// TIA Portal V20 export
FUNCTION_BLOCK "Sequence_1_SemiAutoSplice"   // FB233, LAD
AUTHOR : ERsystem_FA2_DH. Kim
// stored: IsIECCheckEnabled true, MemoryReserve 100, Namespace Unit1.Em2, SetENOAutomatically false
   VAR
      statSelectedJobNumber { ExternalWritable := 'False'} : DInt;   // Evaluated Job Number
      instSequenceLADStatus { ExternalWritable := 'False'} : "LAF_StatusLadSequence";
      instSequenceLADControl { ExternalWritable := 'False'} : "LAF_ControlLadSequence";
      RetryCnt { S7_SetPoint := 'True'} : Array[0..9] of UInt;
      statPulse { ExternalWritable := 'False'} : Array[0..999] of Bool;
      statTonTimer { ExternalWritable := 'False'} : Array[0..9999] of TON_TIME;
   END_VAR
   VAR CONSTANT
      STEP_IDLE : DInt := 1;
      STEP_IMMEDIATE_STOP : DInt := 9001;   // Step executed when an immediate stop command is triggered for the sequence (i.e. when unit is in state aborting)
      SeqDelayTime : Time := T#100ms;
      SeqNoDelayTime : Time;
      RetrySV : UInt := 3;
      JOB_1_STEP_00 : DInt := 100;
      JOB_1_STEP_01 : DInt := 101;
      JOB_1_STEP_02 : DInt := 102;
      JOB_1_STEP_03 : DInt := 103;
      JOB_1_STEP_04 : DInt := 104;
      JOB_1_STEP_05 : DInt := 105;
      JOB_1_STEP_06 : DInt := 106;
      JOB_1_STEP_07 : DInt := 107;
      JOB_1_STEP_08 : DInt := 108;
      JOB_1_STEP_09 : DInt := 109;
      JOB_1_STEP_10 : DInt := 110;
      JOB_1_STEP_11 : DInt := 111;
      JOB_1_STEP_12 : DInt := 112;
      JOB_1_STEP_13 : DInt := 113;
      JOB_1_STEP_14 : DInt := 114;
      JOB_1_STEP_15 : DInt := 115;
      JOB_1_STEP_16 : DInt := 116;
      JOB_1_STEP_17 : DInt := 117;
      JOB_1_STEP_18 : DInt := 118;
      JOB_1_STEP_19 : DInt := 119;
      JOB_1_STEP_20 : DInt := 120;
      JOB_1_STEP_90 : DInt := 190;
      JOB_2_STEP_00 : DInt := 200;
      JOB_2_STEP_01 : DInt := 201;
      JOB_2_STEP_02 : DInt := 202;
      JOB_2_STEP_03 : DInt := 203;
      JOB_2_STEP_04 : DInt := 204;
      JOB_2_STEP_05 : DInt := 205;
      JOB_2_STEP_06 : DInt := 206;
      JOB_2_STEP_07 : DInt := 207;
      JOB_2_STEP_08 : DInt := 208;
      JOB_2_STEP_09 : DInt := 209;
      JOB_2_STEP_10 : DInt := 210;
      JOB_2_STEP_11 : DInt := 211;
      JOB_2_STEP_12 : DInt := 212;
      JOB_2_STEP_13 : DInt := 213;
      JOB_2_STEP_14 : DInt := 214;
      JOB_2_STEP_15 : DInt := 215;
      JOB_2_STEP_16 : DInt := 216;
      JOB_2_STEP_17 : DInt := 217;
      JOB_2_STEP_18 : DInt := 218;
      JOB_2_STEP_19 : DInt := 219;
      JOB_2_STEP_20 : DInt := 220;
      JOB_2_STEP_90 : DInt := 290;
      JOB_3_STEP_00 : DInt := 300;
      JOB_3_STEP_01 : DInt := 301;
      JOB_3_STEP_02 : DInt := 302;
      JOB_3_STEP_03 : DInt := 303;
      JOB_3_STEP_04 : DInt := 304;
      JOB_3_STEP_05 : DInt := 305;
      JOB_3_STEP_06 : DInt := 306;
      JOB_3_STEP_07 : DInt := 307;
      JOB_3_STEP_08 : DInt := 308;
      JOB_3_STEP_09 : DInt := 309;
      JOB_3_STEP_10 : DInt := 310;
      JOB_3_STEP_11 : DInt := 311;
      JOB_3_STEP_12 : DInt := 312;
      JOB_3_STEP_13 : DInt := 313;
      JOB_3_STEP_14 : DInt := 314;
      JOB_3_STEP_15 : DInt := 315;
      JOB_3_STEP_16 : DInt := 316;
      JOB_3_STEP_17 : DInt := 317;
      JOB_3_STEP_18 : DInt := 318;
      JOB_3_STEP_19 : DInt := 319;
      JOB_3_STEP_20 : DInt := 320;
      JOB_3_STEP_90 : DInt := 390;
      JOB_4_STEP_00 : DInt := 400;
      JOB_4_STEP_01 : DInt := 401;
      JOB_4_STEP_02 : DInt := 402;
      JOB_4_STEP_03 : DInt := 403;
      JOB_4_STEP_04 : DInt := 404;
      JOB_4_STEP_05 : DInt := 405;
      JOB_4_STEP_06 : DInt := 406;
      JOB_4_STEP_07 : DInt := 407;
      JOB_4_STEP_08 : DInt := 408;
      JOB_4_STEP_09 : DInt := 409;
      JOB_4_STEP_10 : DInt := 410;
      JOB_4_STEP_11 : DInt := 411;
      JOB_4_STEP_12 : DInt := 412;
      JOB_4_STEP_13 : DInt := 413;
      JOB_4_STEP_14 : DInt := 414;
      JOB_4_STEP_15 : DInt := 415;
      JOB_4_STEP_16 : DInt := 416;
      JOB_4_STEP_17 : DInt := 417;
      JOB_4_STEP_18 : DInt := 418;
      JOB_4_STEP_19 : DInt := 419;
      JOB_4_STEP_20 : DInt := 420;
      JOB_4_STEP_50 : DInt := 450;
      JOB_5_STEP_00 : DInt := 500;
      JOB_5_STEP_01 : DInt := 501;
      JOB_5_STEP_02 : DInt := 502;
      JOB_5_STEP_03 : DInt := 503;
      JOB_5_STEP_04 : DInt := 504;
      JOB_5_STEP_05 : DInt := 505;
      JOB_5_STEP_06 : DInt := 506;
      JOB_5_STEP_07 : DInt := 507;
      JOB_5_STEP_08 : DInt := 508;
      JOB_5_STEP_09 : DInt := 509;
      JOB_5_STEP_10 : DInt := 510;
      JOB_5_STEP_11 : DInt := 511;
      JOB_5_STEP_12 : DInt := 512;
      JOB_5_STEP_13 : DInt := 513;
      JOB_5_STEP_14 : DInt := 514;
      JOB_5_STEP_15 : DInt := 515;
      JOB_5_STEP_16 : DInt := 516;
      JOB_5_STEP_17 : DInt := 517;
      JOB_5_STEP_18 : DInt := 518;
      JOB_5_STEP_19 : DInt := 519;
      JOB_5_STEP_20 : DInt := 520;
      JOB_5_STEP_50 : DInt := 550;
      JOB_6_STEP_00 : DInt := 600;
      JOB_6_STEP_01 : DInt := 601;
      JOB_6_STEP_02 : DInt := 602;
      JOB_6_STEP_03 : DInt := 603;
      JOB_6_STEP_04 : DInt := 604;
      JOB_6_STEP_05 : DInt := 605;
      JOB_6_STEP_06 : DInt := 606;
      JOB_6_STEP_07 : DInt := 607;
      JOB_6_STEP_08 : DInt := 608;
      JOB_6_STEP_09 : DInt := 609;
      JOB_6_STEP_10 : DInt := 610;
      JOB_6_STEP_11 : DInt := 611;
      JOB_6_STEP_12 : DInt := 612;
      JOB_6_STEP_13 : DInt := 613;
      JOB_6_STEP_14 : DInt := 614;
      JOB_6_STEP_15 : DInt := 615;
      JOB_6_STEP_16 : DInt := 616;
      JOB_6_STEP_17 : DInt := 617;
      JOB_6_STEP_18 : DInt := 618;
      JOB_6_STEP_19 : DInt := 619;
      JOB_6_STEP_20 : DInt := 620;
      JOB_6_STEP_50 : DInt := 650;
      JOB_7_STEP_00 : DInt := 700;
      JOB_7_STEP_01 : DInt := 701;
      JOB_7_STEP_02 : DInt := 702;
      JOB_7_STEP_03 : DInt := 703;
      JOB_7_STEP_04 : DInt := 704;
      JOB_7_STEP_05 : DInt := 705;
      JOB_7_STEP_06 : DInt := 706;
      JOB_7_STEP_07 : DInt := 707;
      JOB_7_STEP_08 : DInt := 708;
      JOB_7_STEP_09 : DInt := 709;
      JOB_7_STEP_10 : DInt := 710;
      JOB_7_STEP_11 : DInt := 711;
      JOB_7_STEP_12 : DInt := 712;
      JOB_7_STEP_13 : DInt := 713;
      JOB_7_STEP_14 : DInt := 714;
      JOB_7_STEP_15 : DInt := 715;
      JOB_7_STEP_16 : DInt := 716;
      JOB_7_STEP_17 : DInt := 717;
      JOB_7_STEP_18 : DInt := 718;
      JOB_7_STEP_19 : DInt := 719;
      JOB_7_STEP_20 : DInt := 720;
      JOB_7_STEP_50 : DInt := 750;
      JOB_8_STEP_00 : DInt := 800;
      JOB_8_STEP_01 : DInt := 801;
      JOB_8_STEP_02 : DInt := 802;
      JOB_8_STEP_03 : DInt := 803;
      JOB_8_STEP_04 : DInt := 804;
      JOB_8_STEP_05 : DInt := 805;
      JOB_8_STEP_06 : DInt := 806;
      JOB_8_STEP_07 : DInt := 807;
      JOB_8_STEP_08 : DInt := 808;
      JOB_8_STEP_09 : DInt := 809;
      JOB_8_STEP_10 : DInt := 810;
      JOB_8_STEP_11 : DInt := 811;
      JOB_8_STEP_12 : DInt := 812;
      JOB_8_STEP_13 : DInt := 813;
      JOB_8_STEP_14 : DInt := 814;
      JOB_8_STEP_15 : DInt := 815;
      JOB_8_STEP_16 : DInt := 816;
      JOB_8_STEP_17 : DInt := 817;
      JOB_8_STEP_18 : DInt := 818;
      JOB_8_STEP_19 : DInt := 819;
      JOB_8_STEP_20 : DInt := 820;
      JOB_8_STEP_50 : DInt := 850;
      JOB_9_STEP_00 : DInt := 900;
      JOB_9_STEP_01 : DInt := 901;
      JOB_9_STEP_02 : DInt := 902;
      JOB_9_STEP_03 : DInt := 903;
      JOB_9_STEP_04 : DInt := 904;
      JOB_9_STEP_05 : DInt := 905;
      JOB_9_STEP_06 : DInt := 906;
      JOB_9_STEP_07 : DInt := 907;
      JOB_9_STEP_08 : DInt := 908;
      JOB_9_STEP_09 : DInt := 909;
      JOB_9_STEP_10 : DInt := 910;
      JOB_9_STEP_11 : DInt := 911;
      JOB_9_STEP_12 : DInt := 912;
      JOB_9_STEP_13 : DInt := 913;
      JOB_9_STEP_14 : DInt := 914;
      JOB_9_STEP_15 : DInt := 915;
      JOB_9_STEP_16 : DInt := 916;
      JOB_9_STEP_17 : DInt := 917;
      JOB_9_STEP_18 : DInt := 918;
      JOB_9_STEP_19 : DInt := 919;
      JOB_9_STEP_20 : DInt := 920;
      JOB_8_STEP_51 : DInt := 950;
      JOB_10_STEP_00 : DInt := 1000;
      JOB_10_STEP_01 : DInt := 1001;
      JOB_10_STEP_02 : DInt := 1002;
      JOB_10_STEP_03 : DInt := 1003;
      JOB_10_STEP_04 : DInt := 1004;
      JOB_10_STEP_05 : DInt := 1005;
      JOB_10_STEP_06 : DInt := 1006;
      JOB_10_STEP_07 : DInt := 1007;
      JOB_10_STEP_08 : DInt := 1008;
      JOB_10_STEP_09 : DInt := 1009;
      JOB_10_STEP_10 : DInt := 1010;
      JOB_10_STEP_11 : DInt := 1011;
      JOB_10_STEP_12 : DInt := 1012;
      JOB_10_STEP_13 : DInt := 1013;
      JOB_10_STEP_14 : DInt := 1014;
      JOB_10_STEP_15 : DInt := 1015;
      JOB_10_STEP_16 : DInt := 1016;
      JOB_10_STEP_17 : DInt := 1017;
      JOB_10_STEP_18 : DInt := 1018;
      JOB_10_STEP_19 : DInt := 1019;
      JOB_10_STEP_20 : DInt := 1020;
      JOB_10_STEP_50 : DInt := 1050;
      JOB_11_STEP_00 : DInt := 1100;
      JOB_11_STEP_01 : DInt := 1101;
      JOB_11_STEP_02 : DInt := 1102;
      JOB_11_STEP_03 : DInt := 1103;
      JOB_11_STEP_04 : DInt := 1104;
      JOB_11_STEP_05 : DInt := 1105;
      JOB_11_STEP_06 : DInt := 1106;
      JOB_11_STEP_07 : DInt := 1107;
      JOB_11_STEP_08 : DInt := 1108;
      JOB_11_STEP_09 : DInt := 1109;
      JOB_11_STEP_10 : DInt := 1110;
      JOB_11_STEP_11 : DInt := 1111;
      JOB_11_STEP_12 : DInt := 1112;
      JOB_11_STEP_13 : DInt := 1113;
      JOB_11_STEP_14 : DInt := 1114;
      JOB_11_STEP_15 : DInt := 1115;
      JOB_11_STEP_16 : DInt := 1116;
      JOB_11_STEP_17 : DInt := 1117;
      JOB_11_STEP_18 : DInt := 1118;
      JOB_11_STEP_19 : DInt := 1119;
      JOB_11_STEP_20 : DInt := 1120;
      JOB_11_STEP_50 : DInt := 1150;
      JOB_12_STEP_00 : DInt := 1200;
      JOB_12_STEP_01 : DInt := 1201;
      JOB_12_STEP_02 : DInt := 1202;
      JOB_12_STEP_03 : DInt := 1203;
      JOB_12_STEP_04 : DInt := 1204;
      JOB_12_STEP_05 : DInt := 1205;
      JOB_12_STEP_06 : DInt := 1206;
      JOB_12_STEP_07 : DInt := 1207;
      JOB_12_STEP_08 : DInt := 1208;
      JOB_12_STEP_09 : DInt := 1209;
      JOB_12_STEP_10 : DInt := 1210;
      JOB_12_STEP_11 : DInt := 1211;
      JOB_12_STEP_12 : DInt := 1212;
      JOB_12_STEP_13 : DInt := 1213;
      JOB_12_STEP_14 : DInt := 1214;
      JOB_12_STEP_15 : DInt := 1215;
      JOB_12_STEP_16 : DInt := 1216;
      JOB_12_STEP_17 : DInt := 1217;
      JOB_12_STEP_18 : DInt := 1218;
      JOB_12_STEP_19 : DInt := 1219;
      JOB_12_STEP_20 : DInt := 1220;
      JOB_12_STEP_50 : DInt := 1250;
      JOB_13_STEP_00 : DInt := 1300;
      JOB_13_STEP_01 : DInt := 1301;
      JOB_13_STEP_02 : DInt := 1302;
      JOB_13_STEP_03 : DInt := 1303;
      JOB_13_STEP_04 : DInt := 1304;
      JOB_13_STEP_05 : DInt := 1305;
      JOB_13_STEP_06 : DInt := 1306;
      JOB_13_STEP_07 : DInt := 1307;
      JOB_13_STEP_08 : DInt := 1308;
      JOB_13_STEP_09 : DInt := 1309;
      JOB_13_STEP_10 : DInt := 1310;
      JOB_13_STEP_11 : DInt := 1311;
      JOB_13_STEP_12 : DInt := 1312;
      JOB_13_STEP_13 : DInt := 1313;
      JOB_13_STEP_14 : DInt := 1314;
      JOB_13_STEP_15 : DInt := 1315;
      JOB_13_STEP_16 : DInt := 1316;
      JOB_13_STEP_17 : DInt := 1317;
      JOB_13_STEP_18 : DInt := 1318;
      JOB_13_STEP_19 : DInt := 1319;
      JOB_13_STEP_20 : DInt := 1320;
      JOB_13_STEP_50 : DInt := 1350;
      JOB_14_STEP_00 : DInt := 1400;
      JOB_14_STEP_01 : DInt := 1401;
      JOB_14_STEP_02 : DInt := 1402;
      JOB_14_STEP_03 : DInt := 1403;
      JOB_14_STEP_04 : DInt := 1404;
      JOB_14_STEP_05 : DInt := 1405;
      JOB_14_STEP_06 : DInt := 1406;
      JOB_14_STEP_07 : DInt := 1407;
      JOB_14_STEP_08 : DInt := 1408;
      JOB_14_STEP_09 : DInt := 1409;
      JOB_14_STEP_10 : DInt := 1410;
      JOB_14_STEP_11 : DInt := 1411;
      JOB_14_STEP_12 : DInt := 1412;
      JOB_14_STEP_13 : DInt := 1413;
      JOB_14_STEP_14 : DInt := 1414;
      JOB_14_STEP_15 : DInt := 1415;
      JOB_14_STEP_16 : DInt := 1416;
      JOB_14_STEP_17 : DInt := 1417;
      JOB_14_STEP_18 : DInt := 1418;
      JOB_14_STEP_19 : DInt := 1419;
      JOB_14_STEP_20 : DInt := 1420;
      JOB_14_STEP_50 : DInt := 1450;
      JOB_15_STEP_00 : DInt := 1500;
      JOB_15_STEP_01 : DInt := 1501;
      JOB_15_STEP_02 : DInt := 1502;
      JOB_15_STEP_03 : DInt := 1503;
      JOB_15_STEP_04 : DInt := 1504;
      JOB_15_STEP_05 : DInt := 1505;
      JOB_15_STEP_06 : DInt := 1506;
      JOB_15_STEP_07 : DInt := 1507;
      JOB_15_STEP_08 : DInt := 1508;
      JOB_15_STEP_09 : DInt := 1509;
      JOB_15_STEP_10 : DInt := 1510;
      JOB_15_STEP_11 : DInt := 1511;
      JOB_15_STEP_12 : DInt := 1512;
      JOB_15_STEP_13 : DInt := 1513;
      JOB_15_STEP_14 : DInt := 1514;
      JOB_15_STEP_15 : DInt := 1515;
      JOB_15_STEP_16 : DInt := 1516;
      JOB_15_STEP_17 : DInt := 1517;
      JOB_15_STEP_18 : DInt := 1518;
      JOB_15_STEP_19 : DInt := 1519;
      JOB_15_STEP_20 : DInt := 1520;
      JOB_15_STEP_50 : DInt := 1550;
      JOB_16_STEP_00 : DInt := 1600;
      JOB_16_STEP_01 : DInt := 1601;
      JOB_16_STEP_02 : DInt := 1602;
      JOB_16_STEP_03 : DInt := 1603;
      JOB_16_STEP_04 : DInt := 1604;
      JOB_16_STEP_05 : DInt := 1605;
      JOB_16_STEP_06 : DInt := 1606;
      JOB_16_STEP_07 : DInt := 1607;
      JOB_16_STEP_08 : DInt := 1608;
      JOB_16_STEP_09 : DInt := 1609;
      JOB_16_STEP_10 : DInt := 1610;
      JOB_16_STEP_11 : DInt := 1611;
      JOB_16_STEP_12 : DInt := 1612;
      JOB_16_STEP_13 : DInt := 1613;
      JOB_16_STEP_14 : DInt := 1614;
      JOB_16_STEP_15 : DInt := 1615;
      JOB_16_STEP_16 : DInt := 1616;
      JOB_16_STEP_17 : DInt := 1617;
      JOB_16_STEP_18 : DInt := 1618;
      JOB_16_STEP_19 : DInt := 1619;
      JOB_16_STEP_20 : DInt := 1620;
      JOB_16_STEP_50 : DInt := 1650;
      JOB_17_STEP_00 : DInt := 1700;
      JOB_17_STEP_01 : DInt := 1701;
      JOB_17_STEP_02 : DInt := 1702;
      JOB_17_STEP_03 : DInt := 1703;
      JOB_17_STEP_04 : DInt := 1704;
      JOB_17_STEP_05 : DInt := 1705;
      JOB_17_STEP_06 : DInt := 1706;
      JOB_17_STEP_07 : DInt := 1707;
      JOB_17_STEP_08 : DInt := 1708;
      JOB_17_STEP_09 : DInt := 1709;
      JOB_17_STEP_10 : DInt := 1710;
      JOB_17_STEP_11 : DInt := 1711;
      JOB_17_STEP_12 : DInt := 1712;
      JOB_17_STEP_13 : DInt := 1713;
      JOB_17_STEP_14 : DInt := 1714;
      JOB_17_STEP_15 : DInt := 1715;
      JOB_17_STEP_16 : DInt := 1716;
      JOB_17_STEP_17 : DInt := 1717;
      JOB_17_STEP_18 : DInt := 1718;
      JOB_17_STEP_19 : DInt := 1719;
      JOB_17_STEP_20 : DInt := 1720;
      JOB_17_STEP_50 : DInt := 1750;
      JOB_18_STEP_00 : DInt := 1800;
      JOB_18_STEP_01 : DInt := 1801;
      JOB_18_STEP_02 : DInt := 1802;
      JOB_18_STEP_03 : DInt := 1803;
      JOB_18_STEP_04 : DInt := 1804;
      JOB_18_STEP_05 : DInt := 1805;
      JOB_18_STEP_06 : DInt := 1806;
      JOB_18_STEP_07 : DInt := 1807;
      JOB_18_STEP_08 : DInt := 1808;
      JOB_18_STEP_09 : DInt := 1809;
      JOB_18_STEP_10 : DInt := 1810;
      JOB_18_STEP_11 : DInt := 1811;
      JOB_18_STEP_12 : DInt := 1812;
      JOB_18_STEP_13 : DInt := 1813;
      JOB_18_STEP_14 : DInt := 1814;
      JOB_18_STEP_15 : DInt := 1815;
      JOB_18_STEP_16 : DInt := 1816;
      JOB_18_STEP_17 : DInt := 1817;
      JOB_18_STEP_18 : DInt := 1818;
      JOB_18_STEP_19 : DInt := 1819;
      JOB_18_STEP_20 : DInt := 1820;
      JOB_18_STEP_50 : DInt := 1850;
      JOB_19_STEP_00 : DInt := 1900;
      JOB_19_STEP_01 : DInt := 1901;
      JOB_19_STEP_02 : DInt := 1902;
      JOB_19_STEP_03 : DInt := 1903;
      JOB_19_STEP_04 : DInt := 1904;
      JOB_19_STEP_05 : DInt := 1905;
      JOB_19_STEP_06 : DInt := 1906;
      JOB_19_STEP_07 : DInt := 1907;
      JOB_19_STEP_08 : DInt := 1908;
      JOB_19_STEP_09 : DInt := 1909;
      JOB_19_STEP_10 : DInt := 1910;
      JOB_19_STEP_11 : DInt := 1911;
      JOB_19_STEP_12 : DInt := 1912;
      JOB_19_STEP_13 : DInt := 1913;
      JOB_19_STEP_14 : DInt := 1914;
      JOB_19_STEP_15 : DInt := 1915;
      JOB_19_STEP_16 : DInt := 1916;
      JOB_19_STEP_17 : DInt := 1917;
      JOB_19_STEP_18 : DInt := 1918;
      JOB_19_STEP_19 : DInt := 1919;
      JOB_19_STEP_20 : DInt := 1920;
      JOB_19_STEP_50 : DInt := 1950;
      JOB_20_STEP_00 : DInt := 2000;
      JOB_20_STEP_01 : DInt := 2001;
      JOB_20_STEP_02 : DInt := 2002;
      JOB_20_STEP_03 : DInt := 2003;
      JOB_20_STEP_04 : DInt := 2004;
      JOB_20_STEP_05 : DInt := 2005;
      JOB_20_STEP_06 : DInt := 2006;
      JOB_20_STEP_07 : DInt := 2007;
      JOB_20_STEP_08 : DInt := 2008;
      JOB_20_STEP_09 : DInt := 2009;
      JOB_20_STEP_10 : DInt := 2010;
      JOB_20_STEP_11 : DInt := 2011;
      JOB_20_STEP_12 : DInt := 2012;
      JOB_20_STEP_13 : DInt := 2013;
      JOB_20_STEP_14 : DInt := 2014;
      JOB_20_STEP_15 : DInt := 2015;
      JOB_20_STEP_16 : DInt := 2016;
      JOB_20_STEP_17 : DInt := 2017;
      JOB_20_STEP_18 : DInt := 2018;
      JOB_20_STEP_19 : DInt := 2019;
      JOB_20_STEP_20 : DInt := 2020;
      JOB_20_STEP_50 : DInt := 2050;
      JOB_21_STEP_00 : DInt := 2100;
      JOB_21_STEP_01 : DInt := 2101;
      JOB_21_STEP_02 : DInt := 2102;
      JOB_21_STEP_03 : DInt := 2103;
      JOB_21_STEP_04 : DInt := 2104;
      JOB_21_STEP_05 : DInt := 2105;
      JOB_21_STEP_06 : DInt := 2106;
      JOB_21_STEP_07 : DInt := 2107;
      JOB_21_STEP_08 : DInt := 2108;
      JOB_21_STEP_09 : DInt := 2109;
      JOB_21_STEP_10 : DInt := 2110;
      JOB_21_STEP_11 : DInt := 2111;
      JOB_21_STEP_12 : DInt := 2112;
      JOB_21_STEP_13 : DInt := 2113;
      JOB_21_STEP_14 : DInt := 2114;
      JOB_21_STEP_15 : DInt := 2115;
      JOB_21_STEP_16 : DInt := 2116;
      JOB_21_STEP_17 : DInt := 2117;
      JOB_21_STEP_18 : DInt := 2118;
      JOB_21_STEP_19 : DInt := 2119;
      JOB_21_STEP_20 : DInt := 2120;
      JOB_21_STEP_50 : DInt := 2150;
      JOB_22_STEP_00 : DInt := 2200;
      JOB_22_STEP_01 : DInt := 2201;
      JOB_22_STEP_02 : DInt := 2202;
      JOB_22_STEP_03 : DInt := 2203;
      JOB_22_STEP_04 : DInt := 2204;
      JOB_22_STEP_05 : DInt := 2205;
      JOB_22_STEP_06 : DInt := 2206;
      JOB_22_STEP_07 : DInt := 2207;
      JOB_22_STEP_08 : DInt := 2208;
      JOB_22_STEP_09 : DInt := 2209;
      JOB_22_STEP_10 : DInt := 2210;
      JOB_22_STEP_11 : DInt := 2211;
      JOB_22_STEP_12 : DInt := 2212;
      JOB_22_STEP_13 : DInt := 2213;
      JOB_22_STEP_14 : DInt := 2214;
      JOB_22_STEP_15 : DInt := 2215;
      JOB_22_STEP_16 : DInt := 2216;
      JOB_22_STEP_17 : DInt := 2217;
      JOB_22_STEP_18 : DInt := 2218;
      JOB_22_STEP_19 : DInt := 2219;
      JOB_22_STEP_20 : DInt := 2220;
      JOB_22_STEP_50 : DInt := 2250;
      JOB_23_STEP_00 : DInt := 2300;
      JOB_23_STEP_01 : DInt := 2301;
      JOB_23_STEP_02 : DInt := 2302;
      JOB_23_STEP_03 : DInt := 2303;
      JOB_23_STEP_04 : DInt := 2304;
      JOB_23_STEP_05 : DInt := 2305;
      JOB_23_STEP_06 : DInt := 2306;
      JOB_23_STEP_07 : DInt := 2307;
      JOB_23_STEP_08 : DInt := 2308;
      JOB_23_STEP_09 : DInt := 2309;
      JOB_23_STEP_10 : DInt := 2310;
      JOB_23_STEP_11 : DInt := 2311;
      JOB_23_STEP_12 : DInt := 2312;
      JOB_23_STEP_13 : DInt := 2313;
      JOB_23_STEP_14 : DInt := 2314;
      JOB_23_STEP_15 : DInt := 2315;
      JOB_23_STEP_16 : DInt := 2316;
      JOB_23_STEP_17 : DInt := 2317;
      JOB_23_STEP_18 : DInt := 2318;
      JOB_23_STEP_19 : DInt := 2319;
      JOB_23_STEP_20 : DInt := 2320;
      JOB_23_STEP_50 : DInt := 2350;
      JOB_24_STEP_00 : DInt := 2400;
      JOB_24_STEP_01 : DInt := 2401;
      JOB_24_STEP_02 : DInt := 2402;
      JOB_24_STEP_03 : DInt := 2403;
      JOB_24_STEP_04 : DInt := 2404;
      JOB_24_STEP_05 : DInt := 2405;
      JOB_24_STEP_06 : DInt := 2406;
      JOB_24_STEP_07 : DInt := 2407;
      JOB_24_STEP_08 : DInt := 2408;
      JOB_24_STEP_09 : DInt := 2409;
      JOB_24_STEP_10 : DInt := 2410;
      JOB_24_STEP_11 : DInt := 2411;
      JOB_24_STEP_12 : DInt := 2412;
      JOB_24_STEP_13 : DInt := 2413;
      JOB_24_STEP_14 : DInt := 2414;
      JOB_24_STEP_15 : DInt := 2415;
      JOB_24_STEP_16 : DInt := 2416;
      JOB_24_STEP_17 : DInt := 2417;
      JOB_24_STEP_18 : DInt := 2418;
      JOB_24_STEP_19 : DInt := 2419;
      JOB_24_STEP_20 : DInt := 2420;
      JOB_24_STEP_50 : DInt := 2450;
      JOB_25_STEP_00 : DInt := 2500;
      JOB_25_STEP_01 : DInt := 2501;
      JOB_25_STEP_02 : DInt := 2502;
      JOB_25_STEP_03 : DInt := 2503;
      JOB_25_STEP_04 : DInt := 2504;
      JOB_25_STEP_05 : DInt := 2505;
      JOB_25_STEP_06 : DInt := 2506;
      JOB_25_STEP_07 : DInt := 2507;
      JOB_25_STEP_08 : DInt := 2508;
      JOB_25_STEP_09 : DInt := 2509;
      JOB_25_STEP_10 : DInt := 2510;
      JOB_25_STEP_11 : DInt := 2511;
      JOB_25_STEP_12 : DInt := 2512;
      JOB_25_STEP_13 : DInt := 2513;
      JOB_25_STEP_14 : DInt := 2514;
      JOB_25_STEP_15 : DInt := 2515;
      JOB_25_STEP_16 : DInt := 2516;
      JOB_25_STEP_17 : DInt := 2517;
      JOB_25_STEP_18 : DInt := 2518;
      JOB_25_STEP_19 : DInt := 2519;
      JOB_25_STEP_20 : DInt := 2520;
      JOB_25_STEP_50 : DInt := 2550;
      JOB_26_STEP_00 : DInt := 2600;
      JOB_26_STEP_01 : DInt := 2601;
      JOB_26_STEP_02 : DInt := 2602;
      JOB_26_STEP_03 : DInt := 2603;
      JOB_26_STEP_04 : DInt := 2604;
      JOB_26_STEP_05 : DInt := 2605;
      JOB_26_STEP_06 : DInt := 2606;
      JOB_26_STEP_07 : DInt := 2607;
      JOB_26_STEP_08 : DInt := 2608;
      JOB_26_STEP_09 : DInt := 2609;
      JOB_26_STEP_10 : DInt := 2610;
      JOB_26_STEP_11 : DInt := 2611;
      JOB_26_STEP_12 : DInt := 2612;
      JOB_26_STEP_13 : DInt := 2613;
      JOB_26_STEP_14 : DInt := 2614;
      JOB_26_STEP_15 : DInt := 2615;
      JOB_26_STEP_16 : DInt := 2616;
      JOB_26_STEP_17 : DInt := 2617;
      JOB_26_STEP_18 : DInt := 2618;
      JOB_26_STEP_19 : DInt := 2619;
      JOB_26_STEP_20 : DInt := 2620;
      JOB_26_STEP_50 : DInt := 2650;
      JOB_27_STEP_00 : DInt := 2700;
      JOB_27_STEP_01 : DInt := 2701;
      JOB_27_STEP_02 : DInt := 2702;
      JOB_27_STEP_03 : DInt := 2703;
      JOB_27_STEP_04 : DInt := 2704;
      JOB_27_STEP_05 : DInt := 2705;
      JOB_27_STEP_06 : DInt := 2706;
      JOB_27_STEP_07 : DInt := 2707;
      JOB_27_STEP_08 : DInt := 2708;
      JOB_27_STEP_09 : DInt := 2709;
      JOB_27_STEP_10 : DInt := 2710;
      JOB_27_STEP_11 : DInt := 2711;
      JOB_27_STEP_12 : DInt := 2712;
      JOB_27_STEP_13 : DInt := 2713;
      JOB_27_STEP_14 : DInt := 2714;
      JOB_27_STEP_15 : DInt := 2715;
      JOB_27_STEP_16 : DInt := 2716;
      JOB_27_STEP_17 : DInt := 2717;
      JOB_27_STEP_18 : DInt := 2718;
      JOB_27_STEP_19 : DInt := 2719;
      JOB_27_STEP_20 : DInt := 2720;
      JOB_27_STEP_50 : DInt := 2750;
      JOB_28_STEP_00 : DInt := 2800;
      JOB_28_STEP_01 : DInt := 2801;
      JOB_28_STEP_02 : DInt := 2802;
      JOB_28_STEP_03 : DInt := 2803;
      JOB_28_STEP_04 : DInt := 2804;
      JOB_28_STEP_05 : DInt := 2805;
      JOB_28_STEP_06 : DInt := 2806;
      JOB_28_STEP_07 : DInt := 2807;
      JOB_28_STEP_08 : DInt := 2808;
      JOB_28_STEP_09 : DInt := 2809;
      JOB_28_STEP_10 : DInt := 2810;
      JOB_28_STEP_11 : DInt := 2811;
      JOB_28_STEP_12 : DInt := 2812;
      JOB_28_STEP_13 : DInt := 2813;
      JOB_28_STEP_14 : DInt := 2814;
      JOB_28_STEP_15 : DInt := 2815;
      JOB_28_STEP_16 : DInt := 2816;
      JOB_28_STEP_17 : DInt := 2817;
      JOB_28_STEP_18 : DInt := 2818;
      JOB_28_STEP_19 : DInt := 2819;
      JOB_28_STEP_20 : DInt := 2820;
      JOB_28_STEP_50 : DInt := 2850;
      JOB_29_STEP_00 : DInt := 2900;
      JOB_29_STEP_01 : DInt := 2901;
      JOB_29_STEP_02 : DInt := 2902;
      JOB_29_STEP_03 : DInt := 2903;
      JOB_29_STEP_04 : DInt := 2904;
      JOB_29_STEP_05 : DInt := 2905;
      JOB_29_STEP_06 : DInt := 2906;
      JOB_29_STEP_07 : DInt := 2907;
      JOB_29_STEP_08 : DInt := 2908;
      JOB_29_STEP_09 : DInt := 2909;
      JOB_29_STEP_10 : DInt := 2910;
      JOB_29_STEP_11 : DInt := 2911;
      JOB_29_STEP_12 : DInt := 2912;
      JOB_29_STEP_13 : DInt := 2913;
      JOB_29_STEP_14 : DInt := 2914;
      JOB_29_STEP_15 : DInt := 2915;
      JOB_29_STEP_16 : DInt := 2916;
      JOB_29_STEP_17 : DInt := 2917;
      JOB_29_STEP_18 : DInt := 2918;
      JOB_29_STEP_19 : DInt := 2919;
      JOB_29_STEP_20 : DInt := 2920;
      JOB_29_STEP_50 : DInt := 2950;
      JOB_30_STEP_00 : DInt := 3000;
      JOB_30_STEP_01 : DInt := 3001;
      JOB_30_STEP_02 : DInt := 3002;
      JOB_30_STEP_03 : DInt := 3003;
      JOB_30_STEP_04 : DInt := 3004;
      JOB_30_STEP_05 : DInt := 3005;
      JOB_30_STEP_06 : DInt := 3006;
      JOB_30_STEP_07 : DInt := 3007;
      JOB_30_STEP_08 : DInt := 3008;
      JOB_30_STEP_09 : DInt := 3009;
      JOB_30_STEP_10 : DInt := 3010;
      JOB_30_STEP_11 : DInt := 3011;
      JOB_30_STEP_12 : DInt := 3012;
      JOB_30_STEP_13 : DInt := 3013;
      JOB_30_STEP_14 : DInt := 3014;
      JOB_30_STEP_15 : DInt := 3015;
      JOB_30_STEP_16 : DInt := 3016;
      JOB_30_STEP_17 : DInt := 3017;
      JOB_30_STEP_18 : DInt := 3018;
      JOB_30_STEP_19 : DInt := 3019;
      JOB_30_STEP_20 : DInt := 3020;
      JOB_30_STEP_21 : DInt := 3021;
      JOB_30_STEP_22 : DInt := 3022;
      JOB_30_STEP_23 : DInt := 3023;
      JOB_30_STEP_24 : DInt := 3024;
      JOB_30_STEP_25 : DInt := 3025;
      JOB_30_STEP_26 : DInt := 3026;
      JOB_30_STEP_27 : DInt := 3027;
      JOB_30_STEP_28 : DInt := 3028;
      JOB_30_STEP_29 : DInt := 3029;
      JOB_30_STEP_30 : DInt := 3030;
      JOB_30_STEP_31 : DInt := 3031;
      JOB_30_STEP_32 : DInt := 3032;
      JOB_30_STEP_33 : DInt := 3033;
      JOB_30_STEP_34 : DInt := 3034;
      JOB_30_STEP_35 : DInt := 3035;
      JOB_30_STEP_36 : DInt := 3036;
      JOB_30_STEP_37 : DInt := 3037;
      JOB_30_STEP_38 : DInt := 3038;
      JOB_30_STEP_39 : DInt := 3039;
      JOB_30_STEP_40 : DInt := 3040;
      JOB_30_STEP_41 : DInt := 3041;
      JOB_30_STEP_42 : DInt := 3042;
      JOB_30_STEP_43 : DInt := 3043;
      JOB_30_STEP_44 : DInt := 3044;
      JOB_30_STEP_45 : DInt := 3045;
      JOB_30_STEP_46 : DInt := 3046;
      JOB_30_STEP_47 : DInt := 3047;
      JOB_30_STEP_48 : DInt := 3048;
      JOB_30_STEP_49 : DInt := 3049;
      JOB_30_STEP_50 : DInt := 3050;
      JOB_30_STEP_51 : DInt := 3051;
      JOB_30_STEP_52 : DInt := 3052;
      JOB_30_STEP_53 : DInt := 3053;
      JOB_30_STEP_54 : DInt := 3054;
      JOB_30_STEP_55 : DInt := 3055;
      JOB_30_STEP_56 : DInt := 3056;
      JOB_30_STEP_57 : DInt := 3057;
      JOB_30_STEP_58 : DInt := 3058;
      JOB_30_STEP_59 : DInt := 3059;
      JOB_30_STEP_60 : DInt := 3060;
      JOB_30_STEP_61 : DInt := 3061;
      JOB_30_STEP_62 : DInt := 3062;
      JOB_30_STEP_63 : DInt := 3063;
      JOB_30_STEP_64 : DInt := 3064;
      JOB_30_STEP_65 : DInt := 3065;
      JOB_30_STEP_66 : DInt := 3066;
      JOB_30_STEP_67 : DInt := 3067;
      JOB_30_STEP_68 : DInt := 3068;
      JOB_30_STEP_69 : DInt := 3069;
      JOB_30_STEP_70 : DInt := 3070;
      JOB_30_STEP_71 : DInt := 3071;
      JOB_30_STEP_72 : DInt := 3072;
      JOB_30_STEP_73 : DInt := 3073;
      JOB_30_STEP_74 : DInt := 3074;
      JOB_30_STEP_75 : DInt := 3075;
      JOB_30_STEP_76 : DInt := 3076;
      JOB_30_STEP_77 : DInt := 3077;
      JOB_30_STEP_78 : DInt := 3078;
      JOB_30_STEP_79 : DInt := 3079;
      JOB_30_STEP_80 : DInt := 3080;
      JOB_30_STEP_81 : DInt := 3081;
      JOB_30_STEP_82 : DInt := 3082;
      JOB_30_STEP_83 : DInt := 3083;
      JOB_30_STEP_84 : DInt := 3084;
      JOB_30_STEP_85 : DInt := 3085;
      JOB_30_STEP_86 : DInt := 3086;
      JOB_30_STEP_87 : DInt := 3087;
      JOB_30_STEP_88 : DInt := 3088;
      JOB_30_STEP_89 : DInt := 3089;
      JOB_30_STEP_90 : DInt := 3090;
      JOB_30_STEP_91 : DInt := 3091;
      JOB_30_STEP_92 : DInt := 3092;
      JOB_30_STEP_93 : DInt := 3093;
      JOB_30_STEP_94 : DInt := 3094;
      JOB_30_STEP_95 : DInt := 3095;
      JOB_30_STEP_96 : DInt := 3096;
      JOB_30_STEP_97 : DInt := 3097;
      JOB_30_STEP_98 : DInt := 3098;
      JOB_30_STEP_99 : DInt := 3099;
   END_VAR
   // // RetryCnt[0] : STEP 804
   // // RetryCnt[1] : STEP 1506
   // // RetryCnt[2] : STEP 2506
   // // RetryCnt[3] : STEP 3011
   // // RetryCnt[4] : STEP 3044
   // // RetryCnt[5] : STEP 3081
   VAR_TEMP   // added for the SCL form of the ladder/FBD networks
      _w1 : Bool;
      _w2 : Bool;
   END_VAR
BEGIN

REGION Network 1: BLOCK INFO HEADER
   // (company) / (C) Copyright (year)
   // ---------------------------------------------------------------------------------
   // Title:                             (Title of this block)
   // Comment/Function: (that is implemented in the block)
   // Library/Family:           (that the source is dedicated to)
   // Author:                        (department / person in charge / contact)
   // Target System:          (test system with FW version)
   // Engineering:              TIA Portal (SW version)
   // Restrictions:               (OB types, etc.)
   // Requirements:           (hardware, technological package, etc.)
   // ---------------------------------------------------------------------------------
   // Change log table:
   // Version          | Date             | Signature      | Expert in charge  | Changes applied ------------------------|----------------------|-------------------------|--------------------------------|-----------------------
   // 001.000.000 | yyyy-mm-dd | 0x00000000 | (name of expert) | First released version
END_REGION

REGION Network 2: DESCRIPTION
   // This is a template block provided by the Automation Framework. It can be used to create an own project.
   // The Block Info Header is prepared to put in your own data.
   // Description of the block could be added here and the docu created by Code2Docu.
END_REGION

REGION Network 3: ********************* CONTROL *************************
END_REGION

REGION Network 4: Sequence Control
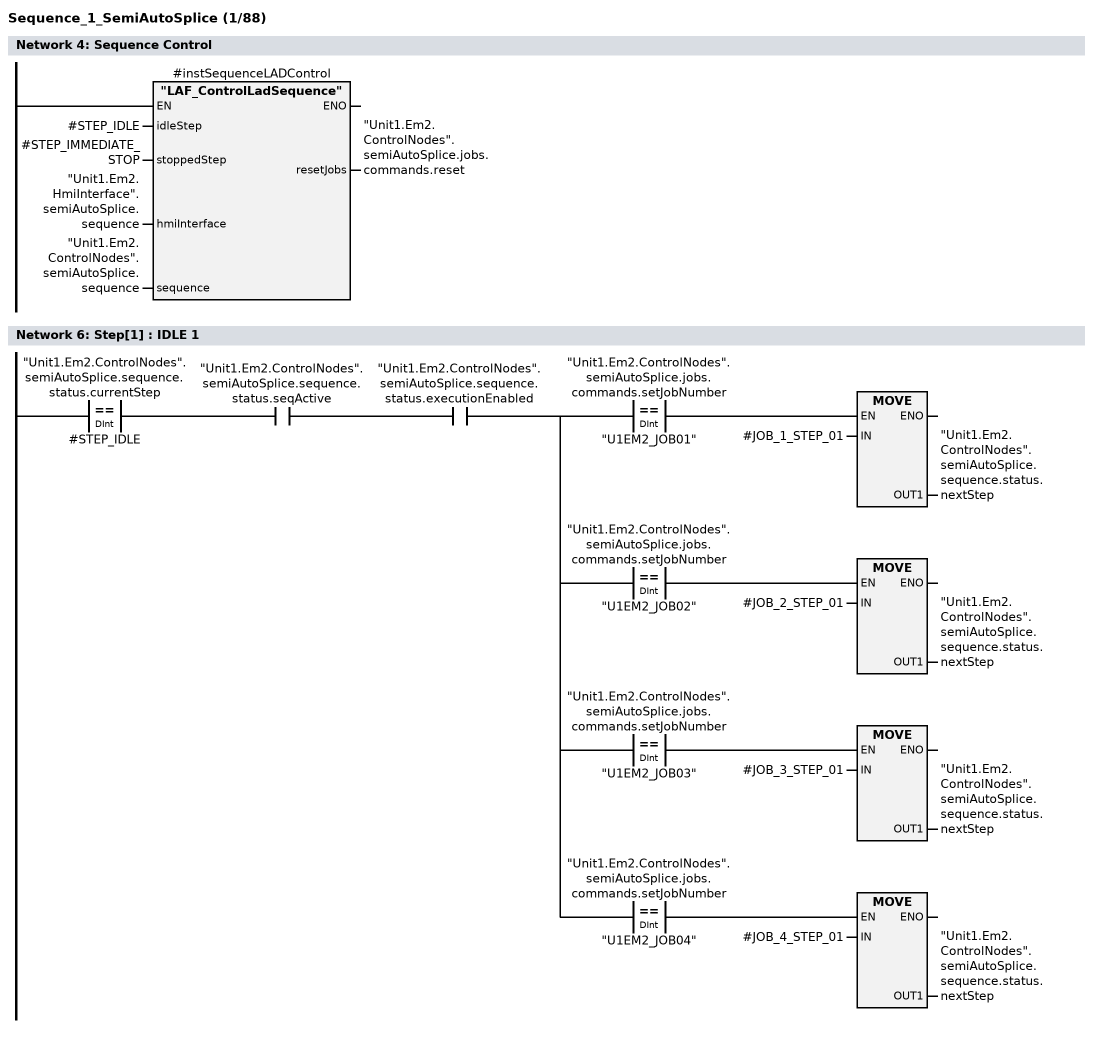
   RUNG wire#powerrail
      #instSequenceLADControl(idleStep := #STEP_IDLE, stoppedStep := #STEP_IMMEDIATE_STOP, hmiInterface := "Unit1.Em2.HmiInterface".semiAutoSplice.sequence, sequence := "Unit1.Em2.ControlNodes".semiAutoSplice.sequence, resetJobs => "Unit1.Em2.ControlNodes".semiAutoSplice.jobs.commands.reset)
   END_RUNG
   // the same network as SCL:
   #instSequenceLADControl(idleStep := #STEP_IDLE,   // "LAF_ControlLadSequence"
                           stoppedStep := #STEP_IMMEDIATE_STOP,
                           hmiInterface := "Unit1.Em2.HmiInterface".semiAutoSplice.sequence,
                           sequence := "Unit1.Em2.ControlNodes".semiAutoSplice.sequence,
                           resetJobs => "Unit1.Em2.ControlNodes".semiAutoSplice.jobs.commands.reset);
END_REGION

REGION Network 6: Step[1] : IDLE 1
   RUNG wire#powerrail
      { S7_Templates := "SrcType := DInt" } EQ_Contact(in1 := "Unit1.Em2.ControlNodes".semiAutoSplice.sequence.status.currentStep, in2 := #STEP_IDLE)
      Contact( "Unit1.Em2.ControlNodes".semiAutoSplice.sequence.status.seqActive )
      Contact( "Unit1.Em2.ControlNodes".semiAutoSplice.sequence.status.executionEnabled )
      wire#w1
      { S7_Templates := "SrcType := DInt" } EQ_Contact(in1 := "Unit1.Em2.ControlNodes".semiAutoSplice.jobs.commands.setJobNumber, in2 := "U1EM2_JOB01")
      Move(in := #JOB_1_STEP_01, out1 => "Unit1.Em2.ControlNodes".semiAutoSplice.sequence.status.nextStep)
   END_RUNG
   RUNG wire#w1
      { S7_Templates := "SrcType := DInt" } EQ_Contact(in1 := "Unit1.Em2.ControlNodes".semiAutoSplice.jobs.commands.setJobNumber, in2 := "U1EM2_JOB02")
      Move(in := #JOB_2_STEP_01, out1 => "Unit1.Em2.ControlNodes".semiAutoSplice.sequence.status.nextStep)
   END_RUNG
   RUNG wire#w1
      { S7_Templates := "SrcType := DInt" } EQ_Contact(in1 := "Unit1.Em2.ControlNodes".semiAutoSplice.jobs.commands.setJobNumber, in2 := "U1EM2_JOB03")
      Move(in := #JOB_3_STEP_01, out1 => "Unit1.Em2.ControlNodes".semiAutoSplice.sequence.status.nextStep)
   END_RUNG
   RUNG wire#w1
      { S7_Templates := "SrcType := DInt" } EQ_Contact(in1 := "Unit1.Em2.ControlNodes".semiAutoSplice.jobs.commands.setJobNumber, in2 := "U1EM2_JOB04")
      Move(in := #JOB_4_STEP_01, out1 => "Unit1.Em2.ControlNodes".semiAutoSplice.sequence.status.nextStep)
   END_RUNG
   // the same network as SCL:
   #_w1 := ("Unit1.Em2.ControlNodes".semiAutoSplice.sequence.status.currentStep = #STEP_IDLE) AND "Unit1.Em2.ControlNodes".semiAutoSplice.sequence.status.seqActive AND "Unit1.Em2.ControlNodes".semiAutoSplice.sequence.status.executionEnabled;
   IF #_w1 AND ("Unit1.Em2.ControlNodes".semiAutoSplice.jobs.commands.setJobNumber = "U1EM2_JOB01") THEN
       "Unit1.Em2.ControlNodes".semiAutoSplice.sequence.status.nextStep := #JOB_1_STEP_01;
   END_IF;
   IF #_w1 AND ("Unit1.Em2.ControlNodes".semiAutoSplice.jobs.commands.setJobNumber = "U1EM2_JOB02") THEN
       "Unit1.Em2.ControlNodes".semiAutoSplice.sequence.status.nextStep := #JOB_2_STEP_01;
   END_IF;
   IF #_w1 AND ("Unit1.Em2.ControlNodes".semiAutoSplice.jobs.commands.setJobNumber = "U1EM2_JOB03") THEN
       "Unit1.Em2.ControlNodes".semiAutoSplice.sequence.status.nextStep := #JOB_3_STEP_01;
   END_IF;
   IF #_w1 AND ("Unit1.Em2.ControlNodes".semiAutoSplice.jobs.commands.setJobNumber = "U1EM2_JOB04") THEN
       "Unit1.Em2.ControlNodes".semiAutoSplice.sequence.status.nextStep := #JOB_4_STEP_01;
   END_IF;
END_REGION

REGION Network 7: Step[1] : IDLE 2
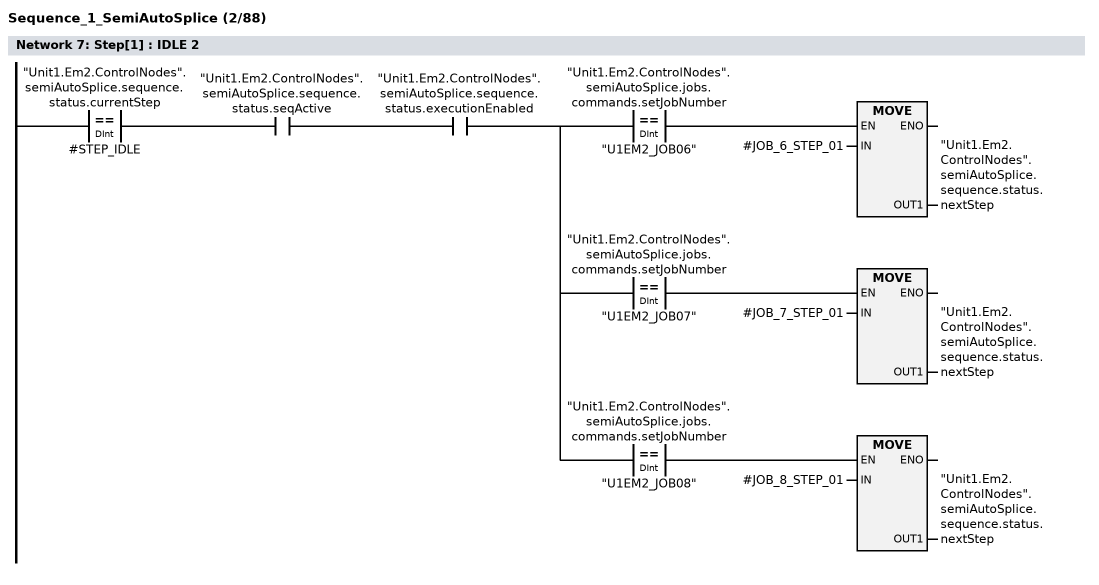
   RUNG wire#powerrail
      { S7_Templates := "SrcType := DInt" } EQ_Contact(in1 := "Unit1.Em2.ControlNodes".semiAutoSplice.sequence.status.currentStep, in2 := #STEP_IDLE)
      Contact( "Unit1.Em2.ControlNodes".semiAutoSplice.sequence.status.seqActive )
      Contact( "Unit1.Em2.ControlNodes".semiAutoSplice.sequence.status.executionEnabled )
      wire#w1
      { S7_Templates := "SrcType := DInt" } EQ_Contact(in1 := "Unit1.Em2.ControlNodes".semiAutoSplice.jobs.commands.setJobNumber, in2 := "U1EM2_JOB06")
      Move(in := #JOB_6_STEP_01, out1 => "Unit1.Em2.ControlNodes".semiAutoSplice.sequence.status.nextStep)
   END_RUNG
   RUNG wire#w1
      { S7_Templates := "SrcType := DInt" } EQ_Contact(in1 := "Unit1.Em2.ControlNodes".semiAutoSplice.jobs.commands.setJobNumber, in2 := "U1EM2_JOB07")
      Move(in := #JOB_7_STEP_01, out1 => "Unit1.Em2.ControlNodes".semiAutoSplice.sequence.status.nextStep)
   END_RUNG
   RUNG wire#w1
      { S7_Templates := "SrcType := DInt" } EQ_Contact(in1 := "Unit1.Em2.ControlNodes".semiAutoSplice.jobs.commands.setJobNumber, in2 := "U1EM2_JOB08")
      Move(in := #JOB_8_STEP_01, out1 => "Unit1.Em2.ControlNodes".semiAutoSplice.sequence.status.nextStep)
   END_RUNG
   // the same network as SCL:
   #_w1 := ("Unit1.Em2.ControlNodes".semiAutoSplice.sequence.status.currentStep = #STEP_IDLE) AND "Unit1.Em2.ControlNodes".semiAutoSplice.sequence.status.seqActive AND "Unit1.Em2.ControlNodes".semiAutoSplice.sequence.status.executionEnabled;
   IF #_w1 AND ("Unit1.Em2.ControlNodes".semiAutoSplice.jobs.commands.setJobNumber = "U1EM2_JOB06") THEN
       "Unit1.Em2.ControlNodes".semiAutoSplice.sequence.status.nextStep := #JOB_6_STEP_01;
   END_IF;
   IF #_w1 AND ("Unit1.Em2.ControlNodes".semiAutoSplice.jobs.commands.setJobNumber = "U1EM2_JOB07") THEN
       "Unit1.Em2.ControlNodes".semiAutoSplice.sequence.status.nextStep := #JOB_7_STEP_01;
   END_IF;
   IF #_w1 AND ("Unit1.Em2.ControlNodes".semiAutoSplice.jobs.commands.setJobNumber = "U1EM2_JOB08") THEN
       "Unit1.Em2.ControlNodes".semiAutoSplice.sequence.status.nextStep := #JOB_8_STEP_01;
   END_IF;
END_REGION

REGION Network 8: Step[1] : IDLE 3
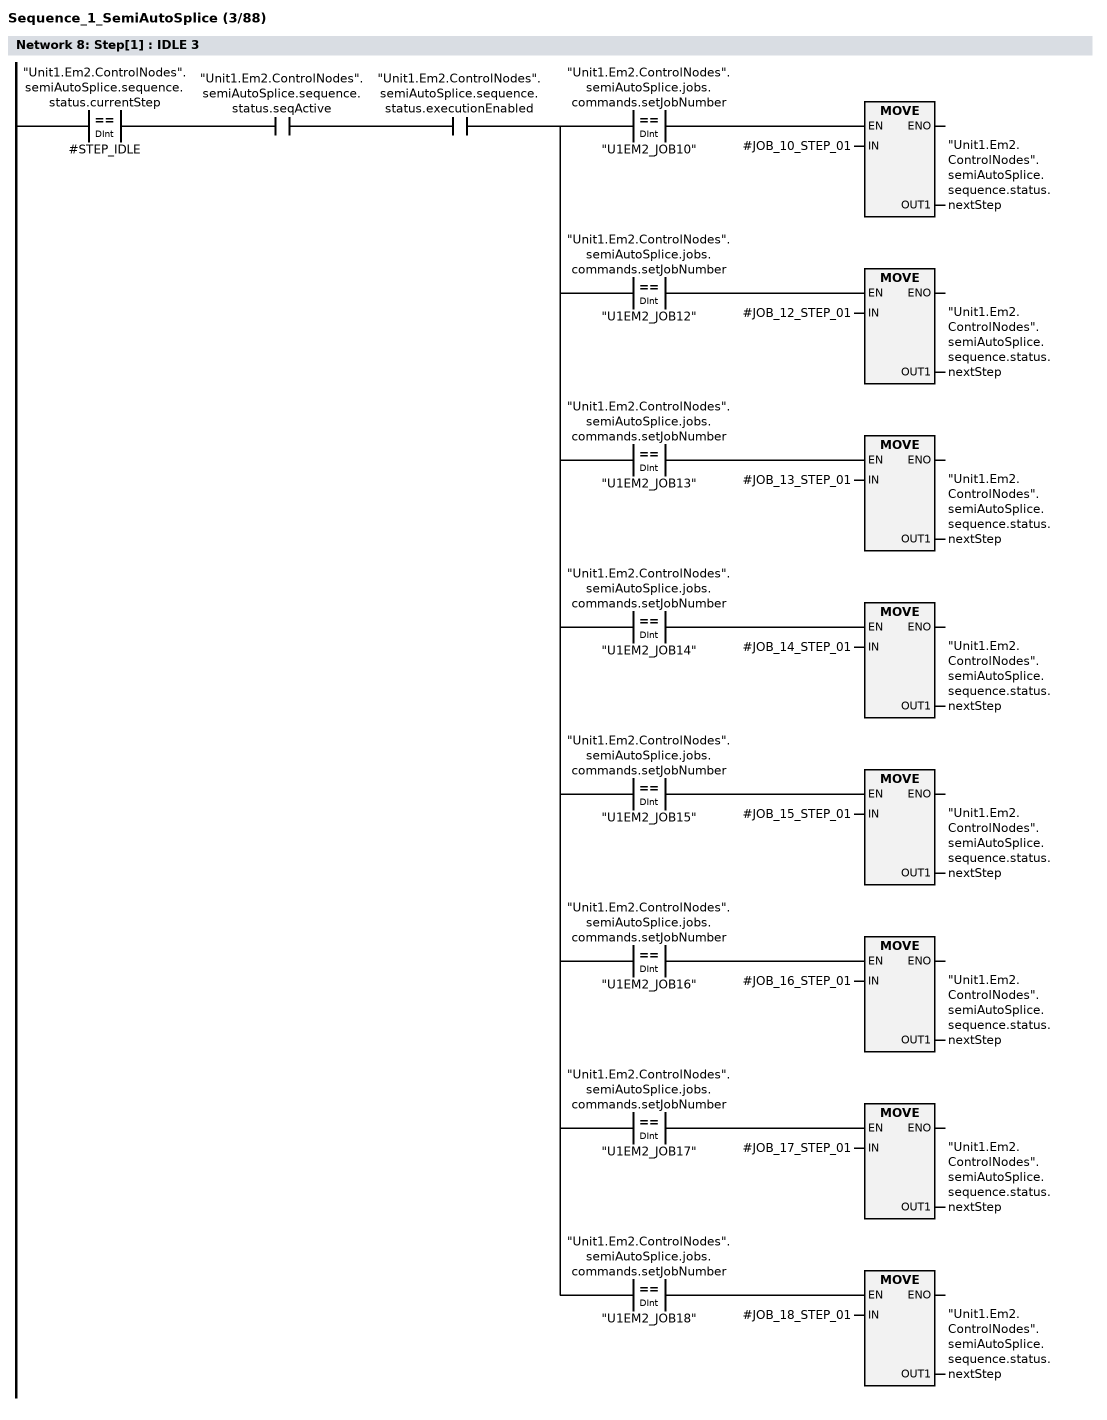
   RUNG wire#powerrail
      { S7_Templates := "SrcType := DInt" } EQ_Contact(in1 := "Unit1.Em2.ControlNodes".semiAutoSplice.sequence.status.currentStep, in2 := #STEP_IDLE)
      Contact( "Unit1.Em2.ControlNodes".semiAutoSplice.sequence.status.seqActive )
      Contact( "Unit1.Em2.ControlNodes".semiAutoSplice.sequence.status.executionEnabled )
      wire#w1
      { S7_Templates := "SrcType := DInt" } EQ_Contact(in1 := "Unit1.Em2.ControlNodes".semiAutoSplice.jobs.commands.setJobNumber, in2 := "U1EM2_JOB10")
      Move(in := #JOB_10_STEP_01, out1 => "Unit1.Em2.ControlNodes".semiAutoSplice.sequence.status.nextStep)
   END_RUNG
   RUNG wire#w1
      { S7_Templates := "SrcType := DInt" } EQ_Contact(in1 := "Unit1.Em2.ControlNodes".semiAutoSplice.jobs.commands.setJobNumber, in2 := "U1EM2_JOB12")
      Move(in := #JOB_12_STEP_01, out1 => "Unit1.Em2.ControlNodes".semiAutoSplice.sequence.status.nextStep)
   END_RUNG
   RUNG wire#w1
      { S7_Templates := "SrcType := DInt" } EQ_Contact(in1 := "Unit1.Em2.ControlNodes".semiAutoSplice.jobs.commands.setJobNumber, in2 := "U1EM2_JOB13")
      Move(in := #JOB_13_STEP_01, out1 => "Unit1.Em2.ControlNodes".semiAutoSplice.sequence.status.nextStep)
   END_RUNG
   RUNG wire#w1
      { S7_Templates := "SrcType := DInt" } EQ_Contact(in1 := "Unit1.Em2.ControlNodes".semiAutoSplice.jobs.commands.setJobNumber, in2 := "U1EM2_JOB14")
      Move(in := #JOB_14_STEP_01, out1 => "Unit1.Em2.ControlNodes".semiAutoSplice.sequence.status.nextStep)
   END_RUNG
   RUNG wire#w1
      { S7_Templates := "SrcType := DInt" } EQ_Contact(in1 := "Unit1.Em2.ControlNodes".semiAutoSplice.jobs.commands.setJobNumber, in2 := "U1EM2_JOB15")
      Move(in := #JOB_15_STEP_01, out1 => "Unit1.Em2.ControlNodes".semiAutoSplice.sequence.status.nextStep)
   END_RUNG
   RUNG wire#w1
      { S7_Templates := "SrcType := DInt" } EQ_Contact(in1 := "Unit1.Em2.ControlNodes".semiAutoSplice.jobs.commands.setJobNumber, in2 := "U1EM2_JOB16")
      Move(in := #JOB_16_STEP_01, out1 => "Unit1.Em2.ControlNodes".semiAutoSplice.sequence.status.nextStep)
   END_RUNG
   RUNG wire#w1
      { S7_Templates := "SrcType := DInt" } EQ_Contact(in1 := "Unit1.Em2.ControlNodes".semiAutoSplice.jobs.commands.setJobNumber, in2 := "U1EM2_JOB17")
      Move(in := #JOB_17_STEP_01, out1 => "Unit1.Em2.ControlNodes".semiAutoSplice.sequence.status.nextStep)
   END_RUNG
   RUNG wire#w1
      { S7_Templates := "SrcType := DInt" } EQ_Contact(in1 := "Unit1.Em2.ControlNodes".semiAutoSplice.jobs.commands.setJobNumber, in2 := "U1EM2_JOB18")
      Move(in := #JOB_18_STEP_01, out1 => "Unit1.Em2.ControlNodes".semiAutoSplice.sequence.status.nextStep)
   END_RUNG
   // the same network as SCL:
   #_w1 := ("Unit1.Em2.ControlNodes".semiAutoSplice.sequence.status.currentStep = #STEP_IDLE) AND "Unit1.Em2.ControlNodes".semiAutoSplice.sequence.status.seqActive AND "Unit1.Em2.ControlNodes".semiAutoSplice.sequence.status.executionEnabled;
   IF #_w1 AND ("Unit1.Em2.ControlNodes".semiAutoSplice.jobs.commands.setJobNumber = "U1EM2_JOB10") THEN
       "Unit1.Em2.ControlNodes".semiAutoSplice.sequence.status.nextStep := #JOB_10_STEP_01;
   END_IF;
   IF #_w1 AND ("Unit1.Em2.ControlNodes".semiAutoSplice.jobs.commands.setJobNumber = "U1EM2_JOB12") THEN
       "Unit1.Em2.ControlNodes".semiAutoSplice.sequence.status.nextStep := #JOB_12_STEP_01;
   END_IF;
   IF #_w1 AND ("Unit1.Em2.ControlNodes".semiAutoSplice.jobs.commands.setJobNumber = "U1EM2_JOB13") THEN
       "Unit1.Em2.ControlNodes".semiAutoSplice.sequence.status.nextStep := #JOB_13_STEP_01;
   END_IF;
   IF #_w1 AND ("Unit1.Em2.ControlNodes".semiAutoSplice.jobs.commands.setJobNumber = "U1EM2_JOB14") THEN
       "Unit1.Em2.ControlNodes".semiAutoSplice.sequence.status.nextStep := #JOB_14_STEP_01;
   END_IF;
   IF #_w1 AND ("Unit1.Em2.ControlNodes".semiAutoSplice.jobs.commands.setJobNumber = "U1EM2_JOB15") THEN
       "Unit1.Em2.ControlNodes".semiAutoSplice.sequence.status.nextStep := #JOB_15_STEP_01;
   END_IF;
   IF #_w1 AND ("Unit1.Em2.ControlNodes".semiAutoSplice.jobs.commands.setJobNumber = "U1EM2_JOB16") THEN
       "Unit1.Em2.ControlNodes".semiAutoSplice.sequence.status.nextStep := #JOB_16_STEP_01;
   END_IF;
   IF #_w1 AND ("Unit1.Em2.ControlNodes".semiAutoSplice.jobs.commands.setJobNumber = "U1EM2_JOB17") THEN
       "Unit1.Em2.ControlNodes".semiAutoSplice.sequence.status.nextStep := #JOB_17_STEP_01;
   END_IF;
   IF #_w1 AND ("Unit1.Em2.ControlNodes".semiAutoSplice.jobs.commands.setJobNumber = "U1EM2_JOB18") THEN
       "Unit1.Em2.ControlNodes".semiAutoSplice.sequence.status.nextStep := #JOB_18_STEP_01;
   END_IF;
END_REGION

REGION Network 9: Step[1] : IDLE 4
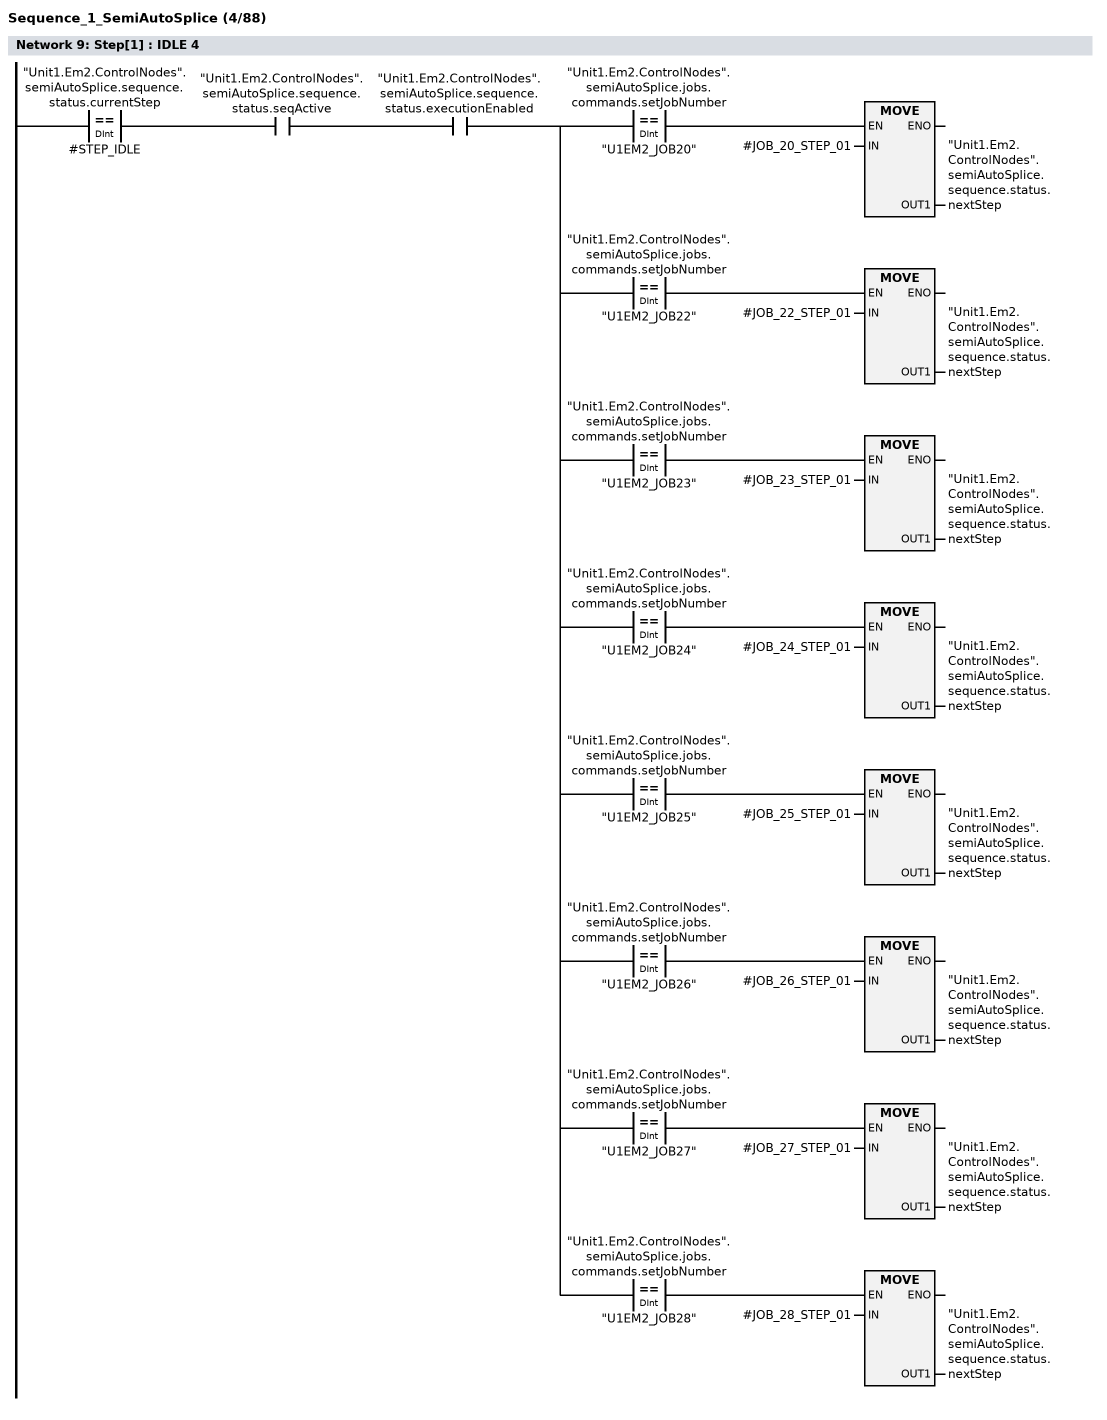
   RUNG wire#powerrail
      { S7_Templates := "SrcType := DInt" } EQ_Contact(in1 := "Unit1.Em2.ControlNodes".semiAutoSplice.sequence.status.currentStep, in2 := #STEP_IDLE)
      Contact( "Unit1.Em2.ControlNodes".semiAutoSplice.sequence.status.seqActive )
      Contact( "Unit1.Em2.ControlNodes".semiAutoSplice.sequence.status.executionEnabled )
      wire#w1
      { S7_Templates := "SrcType := DInt" } EQ_Contact(in1 := "Unit1.Em2.ControlNodes".semiAutoSplice.jobs.commands.setJobNumber, in2 := "U1EM2_JOB20")
      Move(in := #JOB_20_STEP_01, out1 => "Unit1.Em2.ControlNodes".semiAutoSplice.sequence.status.nextStep)
   END_RUNG
   RUNG wire#w1
      { S7_Templates := "SrcType := DInt" } EQ_Contact(in1 := "Unit1.Em2.ControlNodes".semiAutoSplice.jobs.commands.setJobNumber, in2 := "U1EM2_JOB22")
      Move(in := #JOB_22_STEP_01, out1 => "Unit1.Em2.ControlNodes".semiAutoSplice.sequence.status.nextStep)
   END_RUNG
   RUNG wire#w1
      { S7_Templates := "SrcType := DInt" } EQ_Contact(in1 := "Unit1.Em2.ControlNodes".semiAutoSplice.jobs.commands.setJobNumber, in2 := "U1EM2_JOB23")
      Move(in := #JOB_23_STEP_01, out1 => "Unit1.Em2.ControlNodes".semiAutoSplice.sequence.status.nextStep)
   END_RUNG
   RUNG wire#w1
      { S7_Templates := "SrcType := DInt" } EQ_Contact(in1 := "Unit1.Em2.ControlNodes".semiAutoSplice.jobs.commands.setJobNumber, in2 := "U1EM2_JOB24")
      Move(in := #JOB_24_STEP_01, out1 => "Unit1.Em2.ControlNodes".semiAutoSplice.sequence.status.nextStep)
   END_RUNG
   RUNG wire#w1
      { S7_Templates := "SrcType := DInt" } EQ_Contact(in1 := "Unit1.Em2.ControlNodes".semiAutoSplice.jobs.commands.setJobNumber, in2 := "U1EM2_JOB25")
      Move(in := #JOB_25_STEP_01, out1 => "Unit1.Em2.ControlNodes".semiAutoSplice.sequence.status.nextStep)
   END_RUNG
   RUNG wire#w1
      { S7_Templates := "SrcType := DInt" } EQ_Contact(in1 := "Unit1.Em2.ControlNodes".semiAutoSplice.jobs.commands.setJobNumber, in2 := "U1EM2_JOB26")
      Move(in := #JOB_26_STEP_01, out1 => "Unit1.Em2.ControlNodes".semiAutoSplice.sequence.status.nextStep)
   END_RUNG
   RUNG wire#w1
      { S7_Templates := "SrcType := DInt" } EQ_Contact(in1 := "Unit1.Em2.ControlNodes".semiAutoSplice.jobs.commands.setJobNumber, in2 := "U1EM2_JOB27")
      Move(in := #JOB_27_STEP_01, out1 => "Unit1.Em2.ControlNodes".semiAutoSplice.sequence.status.nextStep)
   END_RUNG
   RUNG wire#w1
      { S7_Templates := "SrcType := DInt" } EQ_Contact(in1 := "Unit1.Em2.ControlNodes".semiAutoSplice.jobs.commands.setJobNumber, in2 := "U1EM2_JOB28")
      Move(in := #JOB_28_STEP_01, out1 => "Unit1.Em2.ControlNodes".semiAutoSplice.sequence.status.nextStep)
   END_RUNG
   // the same network as SCL:
   #_w1 := ("Unit1.Em2.ControlNodes".semiAutoSplice.sequence.status.currentStep = #STEP_IDLE) AND "Unit1.Em2.ControlNodes".semiAutoSplice.sequence.status.seqActive AND "Unit1.Em2.ControlNodes".semiAutoSplice.sequence.status.executionEnabled;
   IF #_w1 AND ("Unit1.Em2.ControlNodes".semiAutoSplice.jobs.commands.setJobNumber = "U1EM2_JOB20") THEN
       "Unit1.Em2.ControlNodes".semiAutoSplice.sequence.status.nextStep := #JOB_20_STEP_01;
   END_IF;
   IF #_w1 AND ("Unit1.Em2.ControlNodes".semiAutoSplice.jobs.commands.setJobNumber = "U1EM2_JOB22") THEN
       "Unit1.Em2.ControlNodes".semiAutoSplice.sequence.status.nextStep := #JOB_22_STEP_01;
   END_IF;
   IF #_w1 AND ("Unit1.Em2.ControlNodes".semiAutoSplice.jobs.commands.setJobNumber = "U1EM2_JOB23") THEN
       "Unit1.Em2.ControlNodes".semiAutoSplice.sequence.status.nextStep := #JOB_23_STEP_01;
   END_IF;
   IF #_w1 AND ("Unit1.Em2.ControlNodes".semiAutoSplice.jobs.commands.setJobNumber = "U1EM2_JOB24") THEN
       "Unit1.Em2.ControlNodes".semiAutoSplice.sequence.status.nextStep := #JOB_24_STEP_01;
   END_IF;
   IF #_w1 AND ("Unit1.Em2.ControlNodes".semiAutoSplice.jobs.commands.setJobNumber = "U1EM2_JOB25") THEN
       "Unit1.Em2.ControlNodes".semiAutoSplice.sequence.status.nextStep := #JOB_25_STEP_01;
   END_IF;
   IF #_w1 AND ("Unit1.Em2.ControlNodes".semiAutoSplice.jobs.commands.setJobNumber = "U1EM2_JOB26") THEN
       "Unit1.Em2.ControlNodes".semiAutoSplice.sequence.status.nextStep := #JOB_26_STEP_01;
   END_IF;
   IF #_w1 AND ("Unit1.Em2.ControlNodes".semiAutoSplice.jobs.commands.setJobNumber = "U1EM2_JOB27") THEN
       "Unit1.Em2.ControlNodes".semiAutoSplice.sequence.status.nextStep := #JOB_27_STEP_01;
   END_IF;
   IF #_w1 AND ("Unit1.Em2.ControlNodes".semiAutoSplice.jobs.commands.setJobNumber = "U1EM2_JOB28") THEN
       "Unit1.Em2.ControlNodes".semiAutoSplice.sequence.status.nextStep := #JOB_28_STEP_01;
   END_IF;
END_REGION

REGION Network 10: Step[1] : IDLE 5
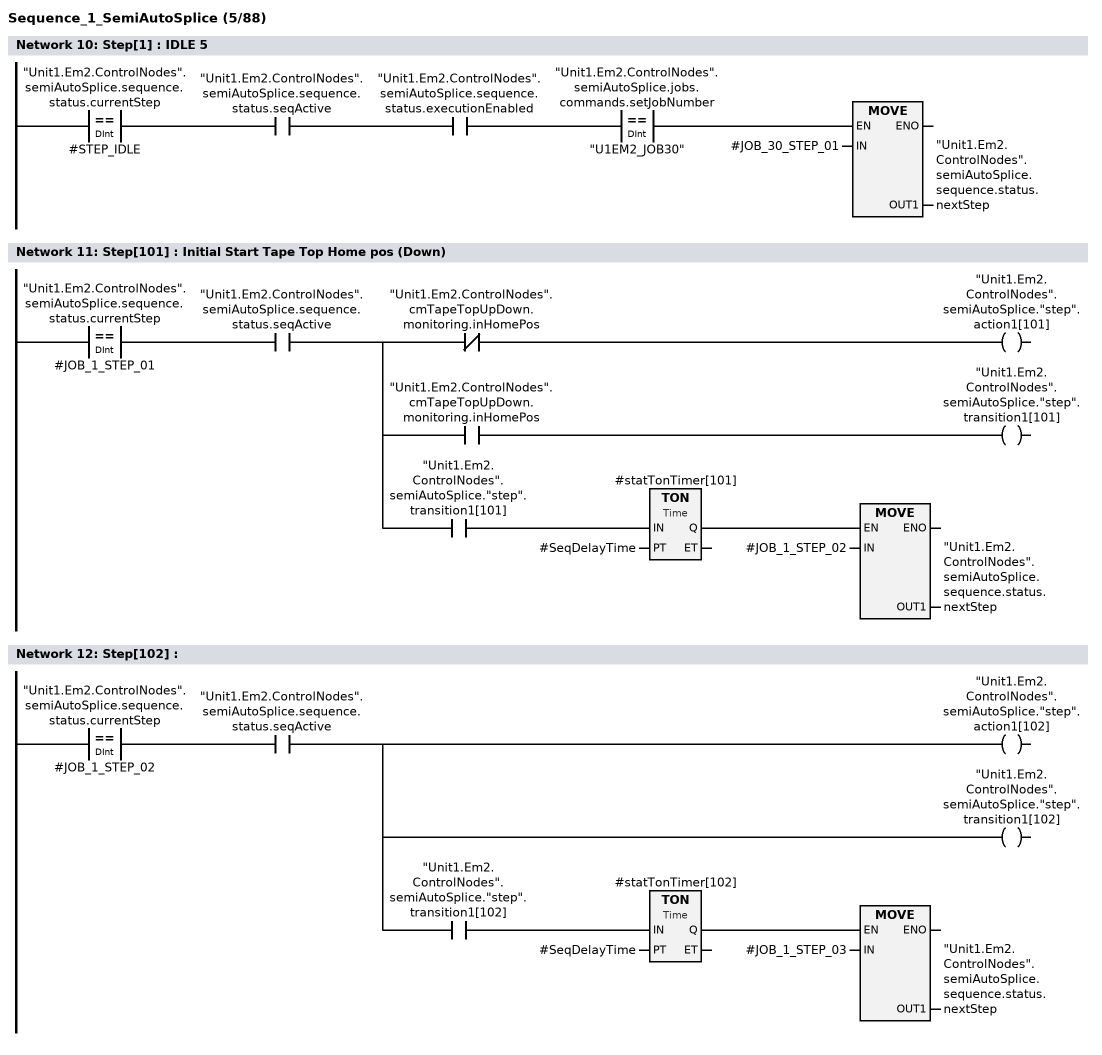
   RUNG wire#powerrail
      { S7_Templates := "SrcType := DInt" } EQ_Contact(in1 := "Unit1.Em2.ControlNodes".semiAutoSplice.sequence.status.currentStep, in2 := #STEP_IDLE)
      Contact( "Unit1.Em2.ControlNodes".semiAutoSplice.sequence.status.seqActive )
      Contact( "Unit1.Em2.ControlNodes".semiAutoSplice.sequence.status.executionEnabled )
      { S7_Templates := "SrcType := DInt" } EQ_Contact(in1 := "Unit1.Em2.ControlNodes".semiAutoSplice.jobs.commands.setJobNumber, in2 := "U1EM2_JOB30")
      Move(in := #JOB_30_STEP_01, out1 => "Unit1.Em2.ControlNodes".semiAutoSplice.sequence.status.nextStep)
   END_RUNG
   // the same network as SCL:
   IF ("Unit1.Em2.ControlNodes".semiAutoSplice.sequence.status.currentStep = #STEP_IDLE) AND "Unit1.Em2.ControlNodes".semiAutoSplice.sequence.status.seqActive AND "Unit1.Em2.ControlNodes".semiAutoSplice.sequence.status.executionEnabled AND ("Unit1.Em2.ControlNodes".semiAutoSplice.jobs.commands.setJobNumber = "U1EM2_JOB30") THEN
       "Unit1.Em2.ControlNodes".semiAutoSplice.sequence.status.nextStep := #JOB_30_STEP_01;
   END_IF;
END_REGION

REGION Network 11: Step[101] : Initial Start Tape Top Home pos (Down)
   RUNG wire#powerrail
      { S7_Templates := "SrcType := DInt" } EQ_Contact(in1 := "Unit1.Em2.ControlNodes".semiAutoSplice.sequence.status.currentStep, in2 := #JOB_1_STEP_01)
      Contact( "Unit1.Em2.ControlNodes".semiAutoSplice.sequence.status.seqActive )
      wire#w1
      I_Contact( "Unit1.Em2.ControlNodes".cmTapeTopUpDown.monitoring.inHomePos )
      Coil( "Unit1.Em2.ControlNodes".semiAutoSplice."step".action1[101] )
   END_RUNG
   RUNG wire#w1
      Contact( "Unit1.Em2.ControlNodes".cmTapeTopUpDown.monitoring.inHomePos )
      Coil( "Unit1.Em2.ControlNodes".semiAutoSplice."step".transition1[101] )
   END_RUNG
   RUNG wire#w1
      Contact( "Unit1.Em2.ControlNodes".semiAutoSplice."step".transition1[101] )
      { S7_Templates := "time_type := Time" } #statTonTimer[101].TON(pt := #SeqDelayTime, et =>)
      Move(in := #JOB_1_STEP_02, out1 => "Unit1.Em2.ControlNodes".semiAutoSplice.sequence.status.nextStep)
   END_RUNG
   // the same network as SCL:
   #_w1 := ("Unit1.Em2.ControlNodes".semiAutoSplice.sequence.status.currentStep = #JOB_1_STEP_01) AND "Unit1.Em2.ControlNodes".semiAutoSplice.sequence.status.seqActive;
   "Unit1.Em2.ControlNodes".semiAutoSplice."step".action1[101] := #_w1 AND NOT "Unit1.Em2.ControlNodes".cmTapeTopUpDown.monitoring.inHomePos;
   "Unit1.Em2.ControlNodes".semiAutoSplice."step".transition1[101] := #_w1 AND "Unit1.Em2.ControlNodes".cmTapeTopUpDown.monitoring.inHomePos;
   #statTonTimer[101].TON(IN := #_w1 AND "Unit1.Em2.ControlNodes".semiAutoSplice."step".transition1[101],
                          PT := #SeqDelayTime);
   IF #statTonTimer[101].Q THEN
       "Unit1.Em2.ControlNodes".semiAutoSplice.sequence.status.nextStep := #JOB_1_STEP_02;
   END_IF;
END_REGION

REGION Network 12: Step[102] :
   RUNG wire#powerrail
      { S7_Templates := "SrcType := DInt" } EQ_Contact(in1 := "Unit1.Em2.ControlNodes".semiAutoSplice.sequence.status.currentStep, in2 := #JOB_1_STEP_02)
      Contact( "Unit1.Em2.ControlNodes".semiAutoSplice.sequence.status.seqActive )
      wire#w1
      Coil( "Unit1.Em2.ControlNodes".semiAutoSplice."step".action1[102] )
   END_RUNG
   RUNG wire#w1
      Coil( "Unit1.Em2.ControlNodes".semiAutoSplice."step".transition1[102] )
   END_RUNG
   RUNG wire#w1
      Contact( "Unit1.Em2.ControlNodes".semiAutoSplice."step".transition1[102] )
      { S7_Templates := "time_type := Time" } #statTonTimer[102].TON(pt := #SeqDelayTime, et =>)
      Move(in := #JOB_1_STEP_03, out1 => "Unit1.Em2.ControlNodes".semiAutoSplice.sequence.status.nextStep)
   END_RUNG
   // the same network as SCL:
   "Unit1.Em2.ControlNodes".semiAutoSplice."step".action1[102] := ("Unit1.Em2.ControlNodes".semiAutoSplice.sequence.status.currentStep = #JOB_1_STEP_02) AND "Unit1.Em2.ControlNodes".semiAutoSplice.sequence.status.seqActive;
   "Unit1.Em2.ControlNodes".semiAutoSplice."step".transition1[102] := ("Unit1.Em2.ControlNodes".semiAutoSplice.sequence.status.currentStep = #JOB_1_STEP_02) AND "Unit1.Em2.ControlNodes".semiAutoSplice.sequence.status.seqActive;
   #statTonTimer[102].TON(IN := ("Unit1.Em2.ControlNodes".semiAutoSplice.sequence.status.currentStep = #JOB_1_STEP_02) AND "Unit1.Em2.ControlNodes".semiAutoSplice.sequence.status.seqActive AND "Unit1.Em2.ControlNodes".semiAutoSplice."step".transition1[102],
                          PT := #SeqDelayTime);
   IF #statTonTimer[102].Q THEN
       "Unit1.Em2.ControlNodes".semiAutoSplice.sequence.status.nextStep := #JOB_1_STEP_03;
   END_IF;
END_REGION

REGION Network 13: Step[103] :
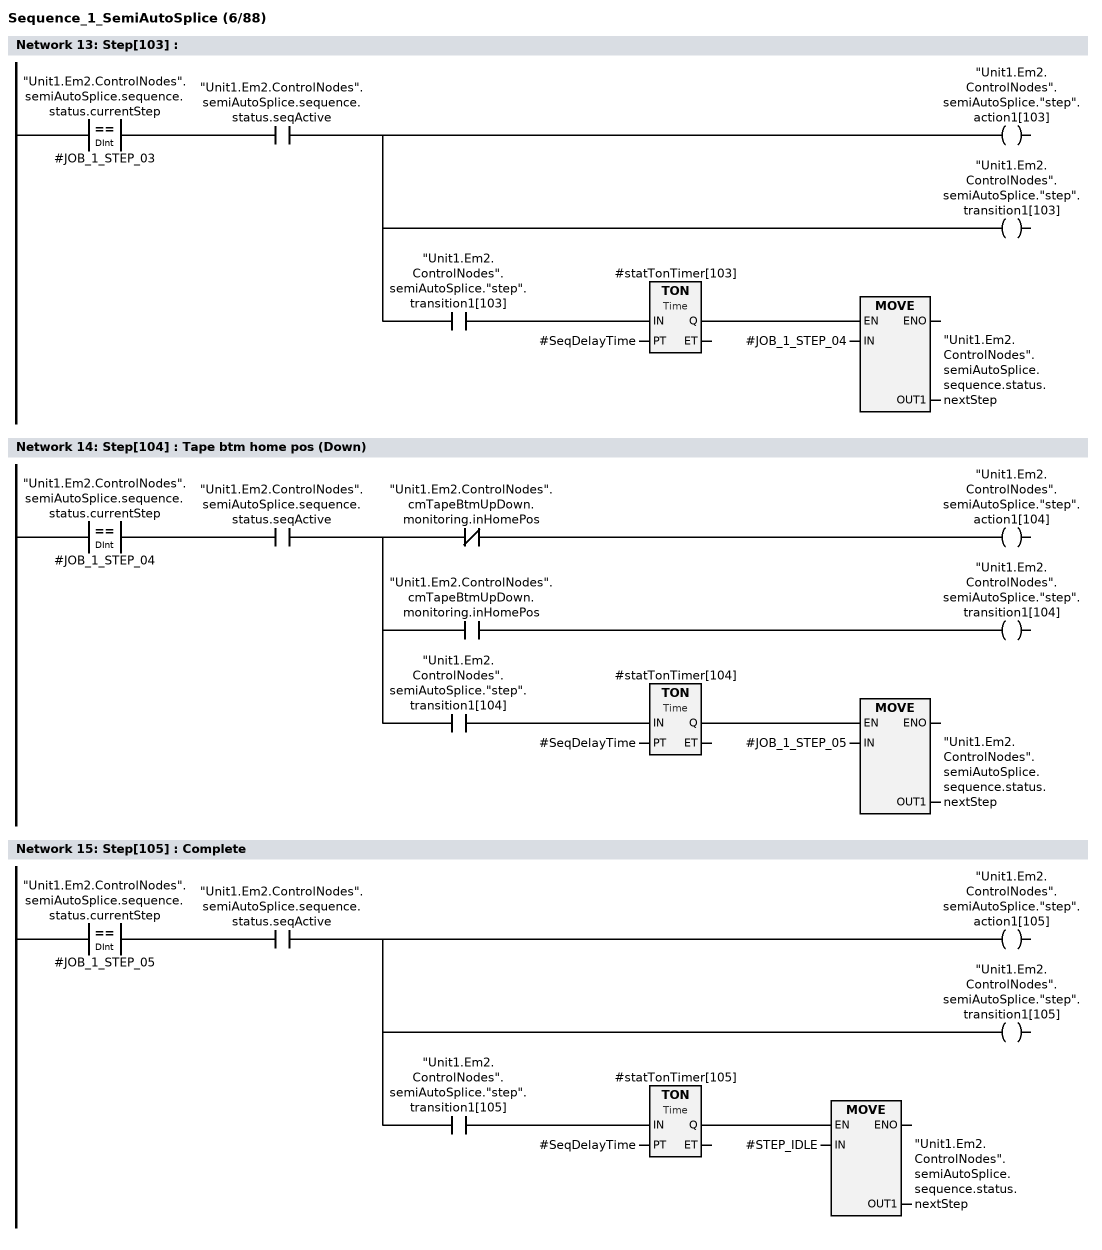
   RUNG wire#powerrail
      { S7_Templates := "SrcType := DInt" } EQ_Contact(in1 := "Unit1.Em2.ControlNodes".semiAutoSplice.sequence.status.currentStep, in2 := #JOB_1_STEP_03)
      Contact( "Unit1.Em2.ControlNodes".semiAutoSplice.sequence.status.seqActive )
      wire#w1
      Coil( "Unit1.Em2.ControlNodes".semiAutoSplice."step".action1[103] )
   END_RUNG
   RUNG wire#w1
      Coil( "Unit1.Em2.ControlNodes".semiAutoSplice."step".transition1[103] )
   END_RUNG
   RUNG wire#w1
      Contact( "Unit1.Em2.ControlNodes".semiAutoSplice."step".transition1[103] )
      { S7_Templates := "time_type := Time" } #statTonTimer[103].TON(pt := #SeqDelayTime, et =>)
      Move(in := #JOB_1_STEP_04, out1 => "Unit1.Em2.ControlNodes".semiAutoSplice.sequence.status.nextStep)
   END_RUNG
   // the same network as SCL:
   "Unit1.Em2.ControlNodes".semiAutoSplice."step".action1[103] := ("Unit1.Em2.ControlNodes".semiAutoSplice.sequence.status.currentStep = #JOB_1_STEP_03) AND "Unit1.Em2.ControlNodes".semiAutoSplice.sequence.status.seqActive;
   "Unit1.Em2.ControlNodes".semiAutoSplice."step".transition1[103] := ("Unit1.Em2.ControlNodes".semiAutoSplice.sequence.status.currentStep = #JOB_1_STEP_03) AND "Unit1.Em2.ControlNodes".semiAutoSplice.sequence.status.seqActive;
   #statTonTimer[103].TON(IN := ("Unit1.Em2.ControlNodes".semiAutoSplice.sequence.status.currentStep = #JOB_1_STEP_03) AND "Unit1.Em2.ControlNodes".semiAutoSplice.sequence.status.seqActive AND "Unit1.Em2.ControlNodes".semiAutoSplice."step".transition1[103],
                          PT := #SeqDelayTime);
   IF #statTonTimer[103].Q THEN
       "Unit1.Em2.ControlNodes".semiAutoSplice.sequence.status.nextStep := #JOB_1_STEP_04;
   END_IF;
END_REGION

REGION Network 14: Step[104] : Tape btm home pos (Down)
   RUNG wire#powerrail
      { S7_Templates := "SrcType := DInt" } EQ_Contact(in1 := "Unit1.Em2.ControlNodes".semiAutoSplice.sequence.status.currentStep, in2 := #JOB_1_STEP_04)
      Contact( "Unit1.Em2.ControlNodes".semiAutoSplice.sequence.status.seqActive )
      wire#w1
      I_Contact( "Unit1.Em2.ControlNodes".cmTapeBtmUpDown.monitoring.inHomePos )
      Coil( "Unit1.Em2.ControlNodes".semiAutoSplice."step".action1[104] )
   END_RUNG
   RUNG wire#w1
      Contact( "Unit1.Em2.ControlNodes".cmTapeBtmUpDown.monitoring.inHomePos )
      Coil( "Unit1.Em2.ControlNodes".semiAutoSplice."step".transition1[104] )
   END_RUNG
   RUNG wire#w1
      Contact( "Unit1.Em2.ControlNodes".semiAutoSplice."step".transition1[104] )
      { S7_Templates := "time_type := Time" } #statTonTimer[104].TON(pt := #SeqDelayTime, et =>)
      Move(in := #JOB_1_STEP_05, out1 => "Unit1.Em2.ControlNodes".semiAutoSplice.sequence.status.nextStep)
   END_RUNG
   // the same network as SCL:
   #_w1 := ("Unit1.Em2.ControlNodes".semiAutoSplice.sequence.status.currentStep = #JOB_1_STEP_04) AND "Unit1.Em2.ControlNodes".semiAutoSplice.sequence.status.seqActive;
   "Unit1.Em2.ControlNodes".semiAutoSplice."step".action1[104] := #_w1 AND NOT "Unit1.Em2.ControlNodes".cmTapeBtmUpDown.monitoring.inHomePos;
   "Unit1.Em2.ControlNodes".semiAutoSplice."step".transition1[104] := #_w1 AND "Unit1.Em2.ControlNodes".cmTapeBtmUpDown.monitoring.inHomePos;
   #statTonTimer[104].TON(IN := #_w1 AND "Unit1.Em2.ControlNodes".semiAutoSplice."step".transition1[104],
                          PT := #SeqDelayTime);
   IF #statTonTimer[104].Q THEN
       "Unit1.Em2.ControlNodes".semiAutoSplice.sequence.status.nextStep := #JOB_1_STEP_05;
   END_IF;
END_REGION

REGION Network 15: Step[105] : Complete
   RUNG wire#powerrail
      { S7_Templates := "SrcType := DInt" } EQ_Contact(in1 := "Unit1.Em2.ControlNodes".semiAutoSplice.sequence.status.currentStep, in2 := #JOB_1_STEP_05)
      Contact( "Unit1.Em2.ControlNodes".semiAutoSplice.sequence.status.seqActive )
      wire#w1
      Coil( "Unit1.Em2.ControlNodes".semiAutoSplice."step".action1[105] )
   END_RUNG
   RUNG wire#w1
      Coil( "Unit1.Em2.ControlNodes".semiAutoSplice."step".transition1[105] )
   END_RUNG
   RUNG wire#w1
      Contact( "Unit1.Em2.ControlNodes".semiAutoSplice."step".transition1[105] )
      { S7_Templates := "time_type := Time" } #statTonTimer[105].TON(pt := #SeqDelayTime, et =>)
      Move(in := #STEP_IDLE, out1 => "Unit1.Em2.ControlNodes".semiAutoSplice.sequence.status.nextStep)
   END_RUNG
   // the same network as SCL:
   "Unit1.Em2.ControlNodes".semiAutoSplice."step".action1[105] := ("Unit1.Em2.ControlNodes".semiAutoSplice.sequence.status.currentStep = #JOB_1_STEP_05) AND "Unit1.Em2.ControlNodes".semiAutoSplice.sequence.status.seqActive;
   "Unit1.Em2.ControlNodes".semiAutoSplice."step".transition1[105] := ("Unit1.Em2.ControlNodes".semiAutoSplice.sequence.status.currentStep = #JOB_1_STEP_05) AND "Unit1.Em2.ControlNodes".semiAutoSplice.sequence.status.seqActive;
   #statTonTimer[105].TON(IN := ("Unit1.Em2.ControlNodes".semiAutoSplice.sequence.status.currentStep = #JOB_1_STEP_05) AND "Unit1.Em2.ControlNodes".semiAutoSplice.sequence.status.seqActive AND "Unit1.Em2.ControlNodes".semiAutoSplice."step".transition1[105],
                          PT := #SeqDelayTime);
   IF #statTonTimer[105].Q THEN
       "Unit1.Em2.ControlNodes".semiAutoSplice.sequence.status.nextStep := #STEP_IDLE;
   END_IF;
END_REGION

REGION Network 16: Step[201] : top & btm Attach home pos Pad Top Home (Down)
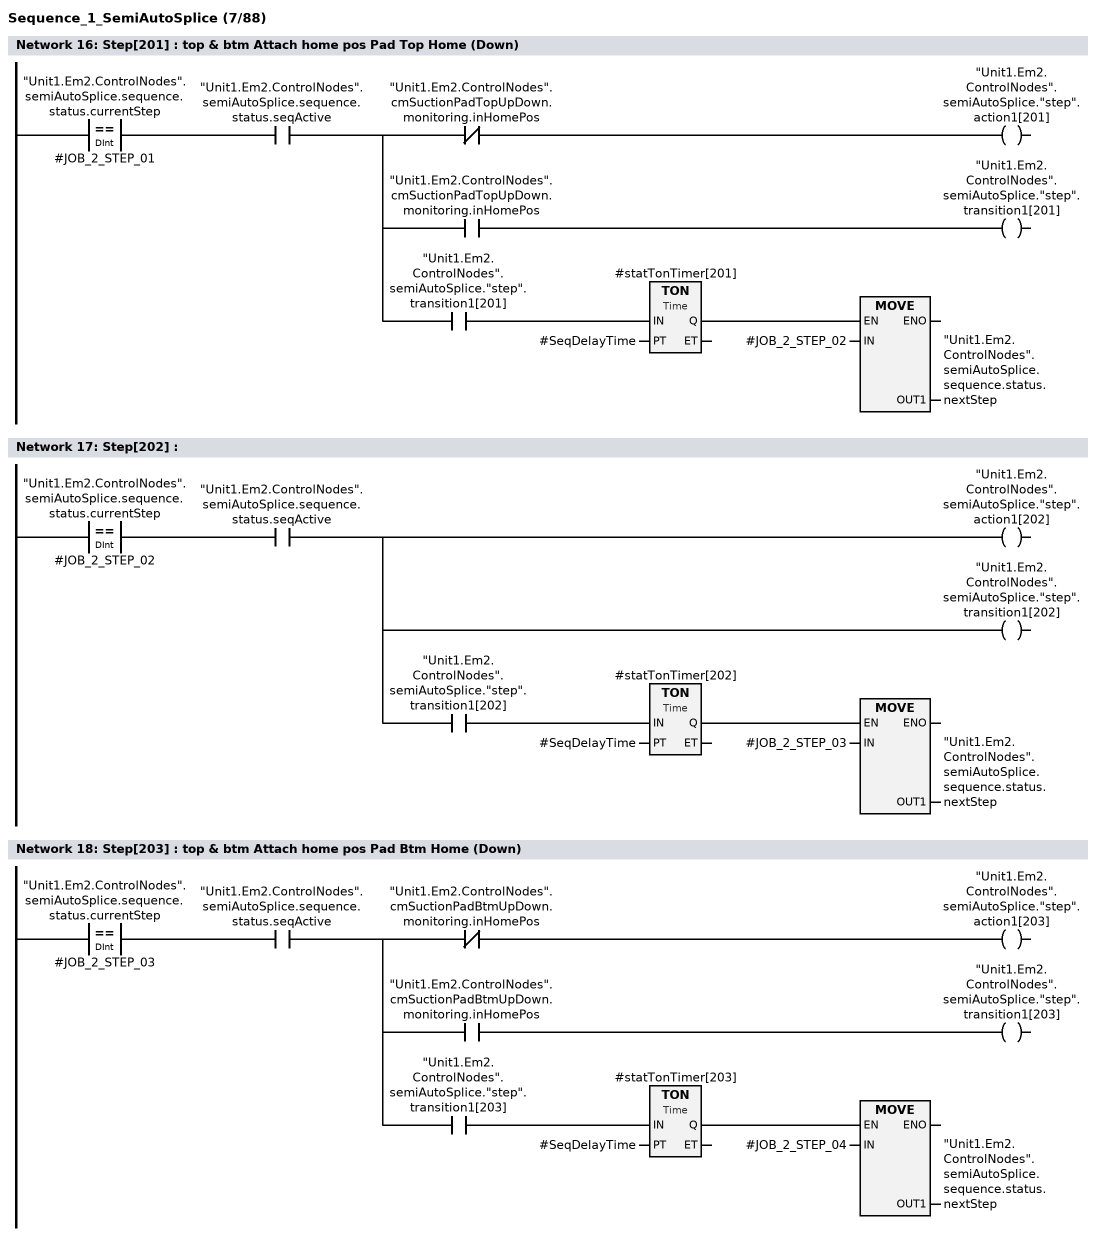
   RUNG wire#powerrail
      { S7_Templates := "SrcType := DInt" } EQ_Contact(in1 := "Unit1.Em2.ControlNodes".semiAutoSplice.sequence.status.currentStep, in2 := #JOB_2_STEP_01)
      Contact( "Unit1.Em2.ControlNodes".semiAutoSplice.sequence.status.seqActive )
      wire#w1
      I_Contact( "Unit1.Em2.ControlNodes".cmSuctionPadTopUpDown.monitoring.inHomePos )
      Coil( "Unit1.Em2.ControlNodes".semiAutoSplice."step".action1[201] )
   END_RUNG
   RUNG wire#w1
      Contact( "Unit1.Em2.ControlNodes".cmSuctionPadTopUpDown.monitoring.inHomePos )
      Coil( "Unit1.Em2.ControlNodes".semiAutoSplice."step".transition1[201] )
   END_RUNG
   RUNG wire#w1
      Contact( "Unit1.Em2.ControlNodes".semiAutoSplice."step".transition1[201] )
      { S7_Templates := "time_type := Time" } #statTonTimer[201].TON(pt := #SeqDelayTime, et =>)
      Move(in := #JOB_2_STEP_02, out1 => "Unit1.Em2.ControlNodes".semiAutoSplice.sequence.status.nextStep)
   END_RUNG
   // the same network as SCL:
   #_w1 := ("Unit1.Em2.ControlNodes".semiAutoSplice.sequence.status.currentStep = #JOB_2_STEP_01) AND "Unit1.Em2.ControlNodes".semiAutoSplice.sequence.status.seqActive;
   "Unit1.Em2.ControlNodes".semiAutoSplice."step".action1[201] := #_w1 AND NOT "Unit1.Em2.ControlNodes".cmSuctionPadTopUpDown.monitoring.inHomePos;
   "Unit1.Em2.ControlNodes".semiAutoSplice."step".transition1[201] := #_w1 AND "Unit1.Em2.ControlNodes".cmSuctionPadTopUpDown.monitoring.inHomePos;
   #statTonTimer[201].TON(IN := #_w1 AND "Unit1.Em2.ControlNodes".semiAutoSplice."step".transition1[201],
                          PT := #SeqDelayTime);
   IF #statTonTimer[201].Q THEN
       "Unit1.Em2.ControlNodes".semiAutoSplice.sequence.status.nextStep := #JOB_2_STEP_02;
   END_IF;
END_REGION

REGION Network 17: Step[202] :
   RUNG wire#powerrail
      { S7_Templates := "SrcType := DInt" } EQ_Contact(in1 := "Unit1.Em2.ControlNodes".semiAutoSplice.sequence.status.currentStep, in2 := #JOB_2_STEP_02)
      Contact( "Unit1.Em2.ControlNodes".semiAutoSplice.sequence.status.seqActive )
      wire#w1
      Coil( "Unit1.Em2.ControlNodes".semiAutoSplice."step".action1[202] )
   END_RUNG
   RUNG wire#w1
      Coil( "Unit1.Em2.ControlNodes".semiAutoSplice."step".transition1[202] )
   END_RUNG
   RUNG wire#w1
      Contact( "Unit1.Em2.ControlNodes".semiAutoSplice."step".transition1[202] )
      { S7_Templates := "time_type := Time" } #statTonTimer[202].TON(pt := #SeqDelayTime, et =>)
      Move(in := #JOB_2_STEP_03, out1 => "Unit1.Em2.ControlNodes".semiAutoSplice.sequence.status.nextStep)
   END_RUNG
   // the same network as SCL:
   "Unit1.Em2.ControlNodes".semiAutoSplice."step".action1[202] := ("Unit1.Em2.ControlNodes".semiAutoSplice.sequence.status.currentStep = #JOB_2_STEP_02) AND "Unit1.Em2.ControlNodes".semiAutoSplice.sequence.status.seqActive;
   "Unit1.Em2.ControlNodes".semiAutoSplice."step".transition1[202] := ("Unit1.Em2.ControlNodes".semiAutoSplice.sequence.status.currentStep = #JOB_2_STEP_02) AND "Unit1.Em2.ControlNodes".semiAutoSplice.sequence.status.seqActive;
   #statTonTimer[202].TON(IN := ("Unit1.Em2.ControlNodes".semiAutoSplice.sequence.status.currentStep = #JOB_2_STEP_02) AND "Unit1.Em2.ControlNodes".semiAutoSplice.sequence.status.seqActive AND "Unit1.Em2.ControlNodes".semiAutoSplice."step".transition1[202],
                          PT := #SeqDelayTime);
   IF #statTonTimer[202].Q THEN
       "Unit1.Em2.ControlNodes".semiAutoSplice.sequence.status.nextStep := #JOB_2_STEP_03;
   END_IF;
END_REGION

REGION Network 18: Step[203] : top & btm Attach home pos Pad Btm Home (Down)
   RUNG wire#powerrail
      { S7_Templates := "SrcType := DInt" } EQ_Contact(in1 := "Unit1.Em2.ControlNodes".semiAutoSplice.sequence.status.currentStep, in2 := #JOB_2_STEP_03)
      Contact( "Unit1.Em2.ControlNodes".semiAutoSplice.sequence.status.seqActive )
      wire#w1
      I_Contact( "Unit1.Em2.ControlNodes".cmSuctionPadBtmUpDown.monitoring.inHomePos )
      Coil( "Unit1.Em2.ControlNodes".semiAutoSplice."step".action1[203] )
   END_RUNG
   RUNG wire#w1
      Contact( "Unit1.Em2.ControlNodes".cmSuctionPadBtmUpDown.monitoring.inHomePos )
      Coil( "Unit1.Em2.ControlNodes".semiAutoSplice."step".transition1[203] )
   END_RUNG
   RUNG wire#w1
      Contact( "Unit1.Em2.ControlNodes".semiAutoSplice."step".transition1[203] )
      { S7_Templates := "time_type := Time" } #statTonTimer[203].TON(pt := #SeqDelayTime, et =>)
      Move(in := #JOB_2_STEP_04, out1 => "Unit1.Em2.ControlNodes".semiAutoSplice.sequence.status.nextStep)
   END_RUNG
   // the same network as SCL:
   #_w1 := ("Unit1.Em2.ControlNodes".semiAutoSplice.sequence.status.currentStep = #JOB_2_STEP_03) AND "Unit1.Em2.ControlNodes".semiAutoSplice.sequence.status.seqActive;
   "Unit1.Em2.ControlNodes".semiAutoSplice."step".action1[203] := #_w1 AND NOT "Unit1.Em2.ControlNodes".cmSuctionPadBtmUpDown.monitoring.inHomePos;
   "Unit1.Em2.ControlNodes".semiAutoSplice."step".transition1[203] := #_w1 AND "Unit1.Em2.ControlNodes".cmSuctionPadBtmUpDown.monitoring.inHomePos;
   #statTonTimer[203].TON(IN := #_w1 AND "Unit1.Em2.ControlNodes".semiAutoSplice."step".transition1[203],
                          PT := #SeqDelayTime);
   IF #statTonTimer[203].Q THEN
       "Unit1.Em2.ControlNodes".semiAutoSplice.sequence.status.nextStep := #JOB_2_STEP_04;
   END_IF;
END_REGION

REGION Network 19: Step[204] :
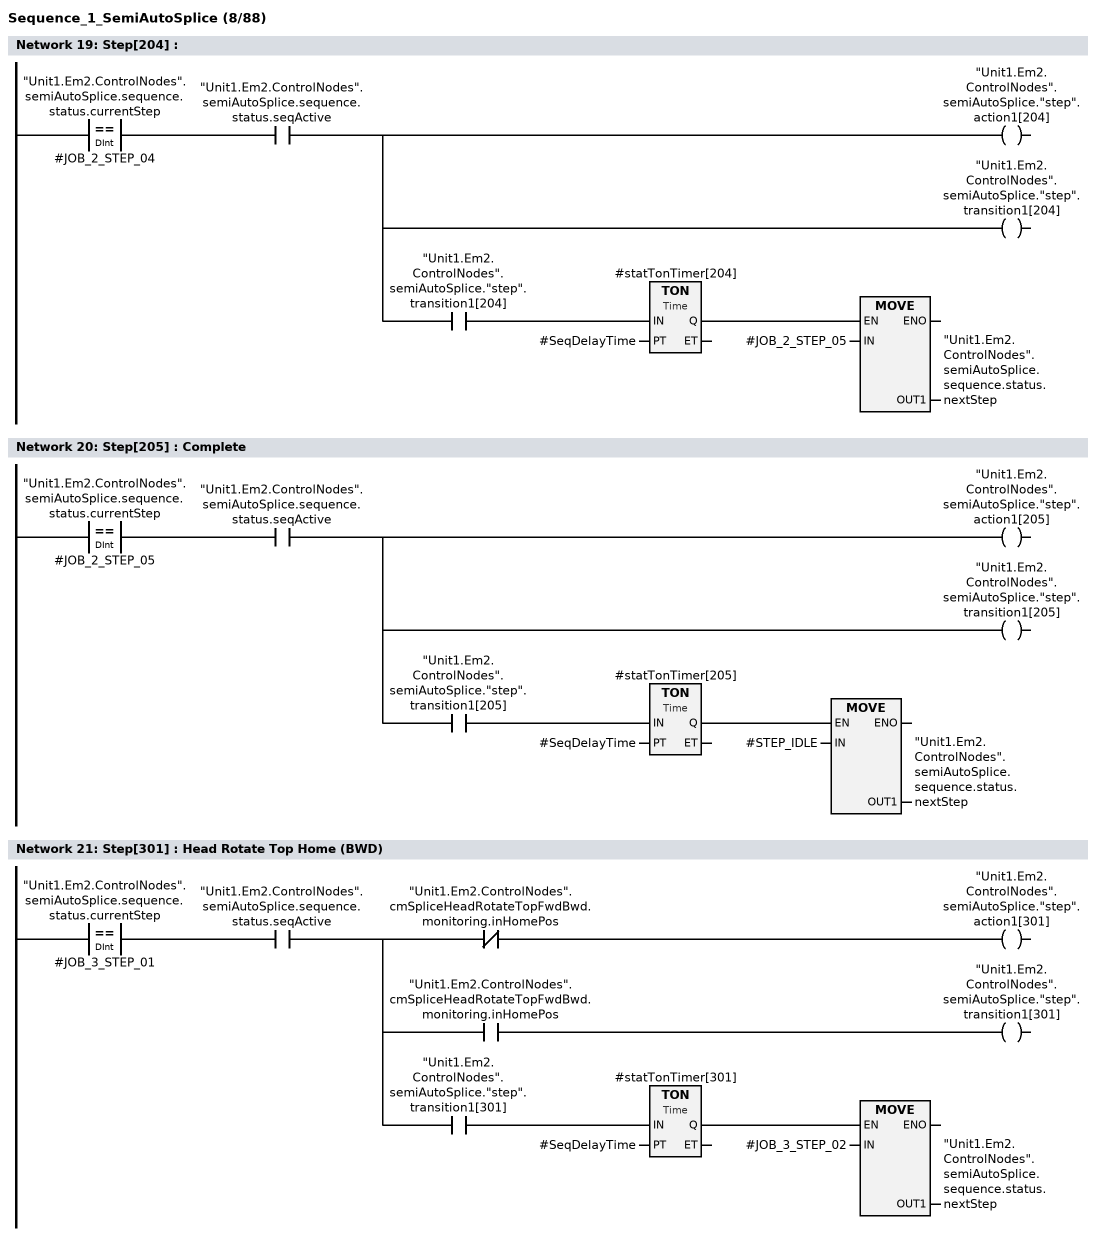
   RUNG wire#powerrail
      { S7_Templates := "SrcType := DInt" } EQ_Contact(in1 := "Unit1.Em2.ControlNodes".semiAutoSplice.sequence.status.currentStep, in2 := #JOB_2_STEP_04)
      Contact( "Unit1.Em2.ControlNodes".semiAutoSplice.sequence.status.seqActive )
      wire#w1
      Coil( "Unit1.Em2.ControlNodes".semiAutoSplice."step".action1[204] )
   END_RUNG
   RUNG wire#w1
      Coil( "Unit1.Em2.ControlNodes".semiAutoSplice."step".transition1[204] )
   END_RUNG
   RUNG wire#w1
      Contact( "Unit1.Em2.ControlNodes".semiAutoSplice."step".transition1[204] )
      { S7_Templates := "time_type := Time" } #statTonTimer[204].TON(pt := #SeqDelayTime, et =>)
      Move(in := #JOB_2_STEP_05, out1 => "Unit1.Em2.ControlNodes".semiAutoSplice.sequence.status.nextStep)
   END_RUNG
   // the same network as SCL:
   "Unit1.Em2.ControlNodes".semiAutoSplice."step".action1[204] := ("Unit1.Em2.ControlNodes".semiAutoSplice.sequence.status.currentStep = #JOB_2_STEP_04) AND "Unit1.Em2.ControlNodes".semiAutoSplice.sequence.status.seqActive;
   "Unit1.Em2.ControlNodes".semiAutoSplice."step".transition1[204] := ("Unit1.Em2.ControlNodes".semiAutoSplice.sequence.status.currentStep = #JOB_2_STEP_04) AND "Unit1.Em2.ControlNodes".semiAutoSplice.sequence.status.seqActive;
   #statTonTimer[204].TON(IN := ("Unit1.Em2.ControlNodes".semiAutoSplice.sequence.status.currentStep = #JOB_2_STEP_04) AND "Unit1.Em2.ControlNodes".semiAutoSplice.sequence.status.seqActive AND "Unit1.Em2.ControlNodes".semiAutoSplice."step".transition1[204],
                          PT := #SeqDelayTime);
   IF #statTonTimer[204].Q THEN
       "Unit1.Em2.ControlNodes".semiAutoSplice.sequence.status.nextStep := #JOB_2_STEP_05;
   END_IF;
END_REGION

REGION Network 20: Step[205] : Complete
   RUNG wire#powerrail
      { S7_Templates := "SrcType := DInt" } EQ_Contact(in1 := "Unit1.Em2.ControlNodes".semiAutoSplice.sequence.status.currentStep, in2 := #JOB_2_STEP_05)
      Contact( "Unit1.Em2.ControlNodes".semiAutoSplice.sequence.status.seqActive )
      wire#w1
      Coil( "Unit1.Em2.ControlNodes".semiAutoSplice."step".action1[205] )
   END_RUNG
   RUNG wire#w1
      Coil( "Unit1.Em2.ControlNodes".semiAutoSplice."step".transition1[205] )
   END_RUNG
   RUNG wire#w1
      Contact( "Unit1.Em2.ControlNodes".semiAutoSplice."step".transition1[205] )
      { S7_Templates := "time_type := Time" } #statTonTimer[205].TON(pt := #SeqDelayTime, et =>)
      Move(in := #STEP_IDLE, out1 => "Unit1.Em2.ControlNodes".semiAutoSplice.sequence.status.nextStep)
   END_RUNG
   // the same network as SCL:
   "Unit1.Em2.ControlNodes".semiAutoSplice."step".action1[205] := ("Unit1.Em2.ControlNodes".semiAutoSplice.sequence.status.currentStep = #JOB_2_STEP_05) AND "Unit1.Em2.ControlNodes".semiAutoSplice.sequence.status.seqActive;
   "Unit1.Em2.ControlNodes".semiAutoSplice."step".transition1[205] := ("Unit1.Em2.ControlNodes".semiAutoSplice.sequence.status.currentStep = #JOB_2_STEP_05) AND "Unit1.Em2.ControlNodes".semiAutoSplice.sequence.status.seqActive;
   #statTonTimer[205].TON(IN := ("Unit1.Em2.ControlNodes".semiAutoSplice.sequence.status.currentStep = #JOB_2_STEP_05) AND "Unit1.Em2.ControlNodes".semiAutoSplice.sequence.status.seqActive AND "Unit1.Em2.ControlNodes".semiAutoSplice."step".transition1[205],
                          PT := #SeqDelayTime);
   IF #statTonTimer[205].Q THEN
       "Unit1.Em2.ControlNodes".semiAutoSplice.sequence.status.nextStep := #STEP_IDLE;
   END_IF;
END_REGION

REGION Network 21: Step[301] : Head Rotate Top Home (BWD)
   RUNG wire#powerrail
      { S7_Templates := "SrcType := DInt" } EQ_Contact(in1 := "Unit1.Em2.ControlNodes".semiAutoSplice.sequence.status.currentStep, in2 := #JOB_3_STEP_01)
      Contact( "Unit1.Em2.ControlNodes".semiAutoSplice.sequence.status.seqActive )
      wire#w1
      I_Contact( "Unit1.Em2.ControlNodes".cmSpliceHeadRotateTopFwdBwd.monitoring.inHomePos )
      Coil( "Unit1.Em2.ControlNodes".semiAutoSplice."step".action1[301] )
   END_RUNG
   RUNG wire#w1
      Contact( "Unit1.Em2.ControlNodes".cmSpliceHeadRotateTopFwdBwd.monitoring.inHomePos )
      Coil( "Unit1.Em2.ControlNodes".semiAutoSplice."step".transition1[301] )
   END_RUNG
   RUNG wire#w1
      Contact( "Unit1.Em2.ControlNodes".semiAutoSplice."step".transition1[301] )
      { S7_Templates := "time_type := Time" } #statTonTimer[301].TON(pt := #SeqDelayTime, et =>)
      Move(in := #JOB_3_STEP_02, out1 => "Unit1.Em2.ControlNodes".semiAutoSplice.sequence.status.nextStep)
   END_RUNG
   // the same network as SCL:
   #_w1 := ("Unit1.Em2.ControlNodes".semiAutoSplice.sequence.status.currentStep = #JOB_3_STEP_01) AND "Unit1.Em2.ControlNodes".semiAutoSplice.sequence.status.seqActive;
   "Unit1.Em2.ControlNodes".semiAutoSplice."step".action1[301] := #_w1 AND NOT "Unit1.Em2.ControlNodes".cmSpliceHeadRotateTopFwdBwd.monitoring.inHomePos;
   "Unit1.Em2.ControlNodes".semiAutoSplice."step".transition1[301] := #_w1 AND "Unit1.Em2.ControlNodes".cmSpliceHeadRotateTopFwdBwd.monitoring.inHomePos;
   #statTonTimer[301].TON(IN := #_w1 AND "Unit1.Em2.ControlNodes".semiAutoSplice."step".transition1[301],
                          PT := #SeqDelayTime);
   IF #statTonTimer[301].Q THEN
       "Unit1.Em2.ControlNodes".semiAutoSplice.sequence.status.nextStep := #JOB_3_STEP_02;
   END_IF;
END_REGION

REGION Network 22: Step[302] :
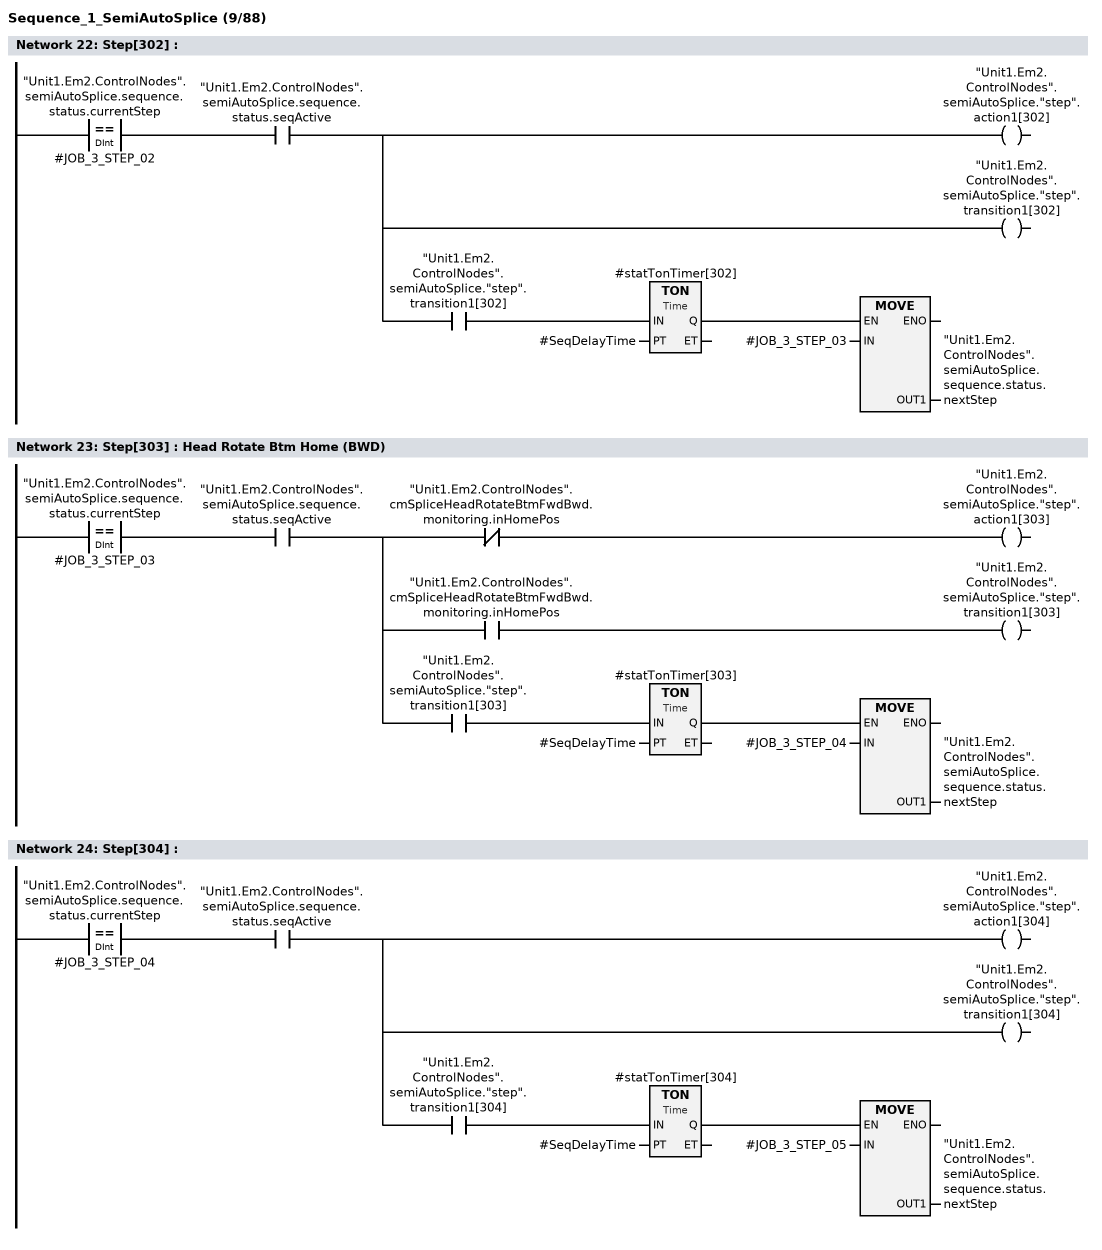
   RUNG wire#powerrail
      { S7_Templates := "SrcType := DInt" } EQ_Contact(in1 := "Unit1.Em2.ControlNodes".semiAutoSplice.sequence.status.currentStep, in2 := #JOB_3_STEP_02)
      Contact( "Unit1.Em2.ControlNodes".semiAutoSplice.sequence.status.seqActive )
      wire#w1
      Coil( "Unit1.Em2.ControlNodes".semiAutoSplice."step".action1[302] )
   END_RUNG
   RUNG wire#w1
      Coil( "Unit1.Em2.ControlNodes".semiAutoSplice."step".transition1[302] )
   END_RUNG
   RUNG wire#w1
      Contact( "Unit1.Em2.ControlNodes".semiAutoSplice."step".transition1[302] )
      { S7_Templates := "time_type := Time" } #statTonTimer[302].TON(pt := #SeqDelayTime, et =>)
      Move(in := #JOB_3_STEP_03, out1 => "Unit1.Em2.ControlNodes".semiAutoSplice.sequence.status.nextStep)
   END_RUNG
   // the same network as SCL:
   "Unit1.Em2.ControlNodes".semiAutoSplice."step".action1[302] := ("Unit1.Em2.ControlNodes".semiAutoSplice.sequence.status.currentStep = #JOB_3_STEP_02) AND "Unit1.Em2.ControlNodes".semiAutoSplice.sequence.status.seqActive;
   "Unit1.Em2.ControlNodes".semiAutoSplice."step".transition1[302] := ("Unit1.Em2.ControlNodes".semiAutoSplice.sequence.status.currentStep = #JOB_3_STEP_02) AND "Unit1.Em2.ControlNodes".semiAutoSplice.sequence.status.seqActive;
   #statTonTimer[302].TON(IN := ("Unit1.Em2.ControlNodes".semiAutoSplice.sequence.status.currentStep = #JOB_3_STEP_02) AND "Unit1.Em2.ControlNodes".semiAutoSplice.sequence.status.seqActive AND "Unit1.Em2.ControlNodes".semiAutoSplice."step".transition1[302],
                          PT := #SeqDelayTime);
   IF #statTonTimer[302].Q THEN
       "Unit1.Em2.ControlNodes".semiAutoSplice.sequence.status.nextStep := #JOB_3_STEP_03;
   END_IF;
END_REGION

REGION Network 23: Step[303] : Head Rotate Btm Home (BWD)
   RUNG wire#powerrail
      { S7_Templates := "SrcType := DInt" } EQ_Contact(in1 := "Unit1.Em2.ControlNodes".semiAutoSplice.sequence.status.currentStep, in2 := #JOB_3_STEP_03)
      Contact( "Unit1.Em2.ControlNodes".semiAutoSplice.sequence.status.seqActive )
      wire#w1
      I_Contact( "Unit1.Em2.ControlNodes".cmSpliceHeadRotateBtmFwdBwd.monitoring.inHomePos )
      Coil( "Unit1.Em2.ControlNodes".semiAutoSplice."step".action1[303] )
   END_RUNG
   RUNG wire#w1
      Contact( "Unit1.Em2.ControlNodes".cmSpliceHeadRotateBtmFwdBwd.monitoring.inHomePos )
      Coil( "Unit1.Em2.ControlNodes".semiAutoSplice."step".transition1[303] )
   END_RUNG
   RUNG wire#w1
      Contact( "Unit1.Em2.ControlNodes".semiAutoSplice."step".transition1[303] )
      { S7_Templates := "time_type := Time" } #statTonTimer[303].TON(pt := #SeqDelayTime, et =>)
      Move(in := #JOB_3_STEP_04, out1 => "Unit1.Em2.ControlNodes".semiAutoSplice.sequence.status.nextStep)
   END_RUNG
   // the same network as SCL:
   #_w1 := ("Unit1.Em2.ControlNodes".semiAutoSplice.sequence.status.currentStep = #JOB_3_STEP_03) AND "Unit1.Em2.ControlNodes".semiAutoSplice.sequence.status.seqActive;
   "Unit1.Em2.ControlNodes".semiAutoSplice."step".action1[303] := #_w1 AND NOT "Unit1.Em2.ControlNodes".cmSpliceHeadRotateBtmFwdBwd.monitoring.inHomePos;
   "Unit1.Em2.ControlNodes".semiAutoSplice."step".transition1[303] := #_w1 AND "Unit1.Em2.ControlNodes".cmSpliceHeadRotateBtmFwdBwd.monitoring.inHomePos;
   #statTonTimer[303].TON(IN := #_w1 AND "Unit1.Em2.ControlNodes".semiAutoSplice."step".transition1[303],
                          PT := #SeqDelayTime);
   IF #statTonTimer[303].Q THEN
       "Unit1.Em2.ControlNodes".semiAutoSplice.sequence.status.nextStep := #JOB_3_STEP_04;
   END_IF;
END_REGION

REGION Network 24: Step[304] :
   RUNG wire#powerrail
      { S7_Templates := "SrcType := DInt" } EQ_Contact(in1 := "Unit1.Em2.ControlNodes".semiAutoSplice.sequence.status.currentStep, in2 := #JOB_3_STEP_04)
      Contact( "Unit1.Em2.ControlNodes".semiAutoSplice.sequence.status.seqActive )
      wire#w1
      Coil( "Unit1.Em2.ControlNodes".semiAutoSplice."step".action1[304] )
   END_RUNG
   RUNG wire#w1
      Coil( "Unit1.Em2.ControlNodes".semiAutoSplice."step".transition1[304] )
   END_RUNG
   RUNG wire#w1
      Contact( "Unit1.Em2.ControlNodes".semiAutoSplice."step".transition1[304] )
      { S7_Templates := "time_type := Time" } #statTonTimer[304].TON(pt := #SeqDelayTime, et =>)
      Move(in := #JOB_3_STEP_05, out1 => "Unit1.Em2.ControlNodes".semiAutoSplice.sequence.status.nextStep)
   END_RUNG
   // the same network as SCL:
   "Unit1.Em2.ControlNodes".semiAutoSplice."step".action1[304] := ("Unit1.Em2.ControlNodes".semiAutoSplice.sequence.status.currentStep = #JOB_3_STEP_04) AND "Unit1.Em2.ControlNodes".semiAutoSplice.sequence.status.seqActive;
   "Unit1.Em2.ControlNodes".semiAutoSplice."step".transition1[304] := ("Unit1.Em2.ControlNodes".semiAutoSplice.sequence.status.currentStep = #JOB_3_STEP_04) AND "Unit1.Em2.ControlNodes".semiAutoSplice.sequence.status.seqActive;
   #statTonTimer[304].TON(IN := ("Unit1.Em2.ControlNodes".semiAutoSplice.sequence.status.currentStep = #JOB_3_STEP_04) AND "Unit1.Em2.ControlNodes".semiAutoSplice.sequence.status.seqActive AND "Unit1.Em2.ControlNodes".semiAutoSplice."step".transition1[304],
                          PT := #SeqDelayTime);
   IF #statTonTimer[304].Q THEN
       "Unit1.Em2.ControlNodes".semiAutoSplice.sequence.status.nextStep := #JOB_3_STEP_05;
   END_IF;
END_REGION

REGION Network 25: Step[305] : Complete
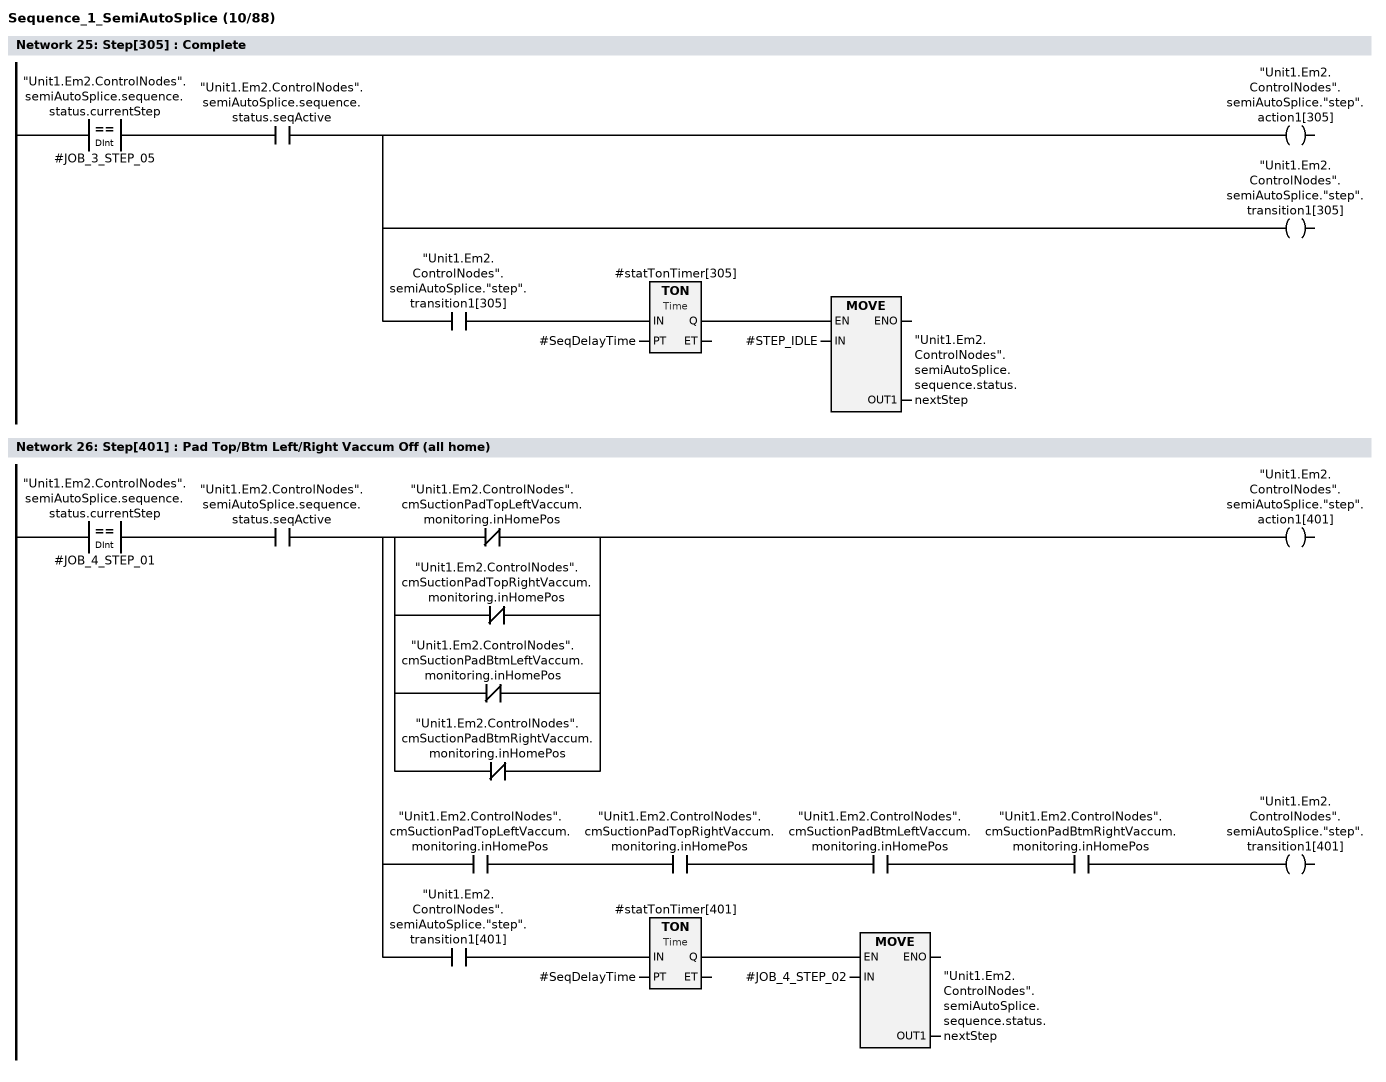
   RUNG wire#powerrail
      { S7_Templates := "SrcType := DInt" } EQ_Contact(in1 := "Unit1.Em2.ControlNodes".semiAutoSplice.sequence.status.currentStep, in2 := #JOB_3_STEP_05)
      Contact( "Unit1.Em2.ControlNodes".semiAutoSplice.sequence.status.seqActive )
      wire#w1
      Coil( "Unit1.Em2.ControlNodes".semiAutoSplice."step".action1[305] )
   END_RUNG
   RUNG wire#w1
      Coil( "Unit1.Em2.ControlNodes".semiAutoSplice."step".transition1[305] )
   END_RUNG
   RUNG wire#w1
      Contact( "Unit1.Em2.ControlNodes".semiAutoSplice."step".transition1[305] )
      { S7_Templates := "time_type := Time" } #statTonTimer[305].TON(pt := #SeqDelayTime, et =>)
      Move(in := #STEP_IDLE, out1 => "Unit1.Em2.ControlNodes".semiAutoSplice.sequence.status.nextStep)
   END_RUNG
   // the same network as SCL:
   "Unit1.Em2.ControlNodes".semiAutoSplice."step".action1[305] := ("Unit1.Em2.ControlNodes".semiAutoSplice.sequence.status.currentStep = #JOB_3_STEP_05) AND "Unit1.Em2.ControlNodes".semiAutoSplice.sequence.status.seqActive;
   "Unit1.Em2.ControlNodes".semiAutoSplice."step".transition1[305] := ("Unit1.Em2.ControlNodes".semiAutoSplice.sequence.status.currentStep = #JOB_3_STEP_05) AND "Unit1.Em2.ControlNodes".semiAutoSplice.sequence.status.seqActive;
   #statTonTimer[305].TON(IN := ("Unit1.Em2.ControlNodes".semiAutoSplice.sequence.status.currentStep = #JOB_3_STEP_05) AND "Unit1.Em2.ControlNodes".semiAutoSplice.sequence.status.seqActive AND "Unit1.Em2.ControlNodes".semiAutoSplice."step".transition1[305],
                          PT := #SeqDelayTime);
   IF #statTonTimer[305].Q THEN
       "Unit1.Em2.ControlNodes".semiAutoSplice.sequence.status.nextStep := #STEP_IDLE;
   END_IF;
END_REGION

REGION Network 26: Step[401] : Pad Top/Btm Left/Right Vaccum Off (all home)
   RUNG wire#powerrail
      { S7_Templates := "SrcType := DInt" } EQ_Contact(in1 := "Unit1.Em2.ControlNodes".semiAutoSplice.sequence.status.currentStep, in2 := #JOB_4_STEP_01)
      Contact( "Unit1.Em2.ControlNodes".semiAutoSplice.sequence.status.seqActive )
      wire#w1
      I_Contact( "Unit1.Em2.ControlNodes".cmSuctionPadTopLeftVaccum.monitoring.inHomePos )
      wire#w2
      Coil( "Unit1.Em2.ControlNodes".semiAutoSplice."step".action1[401] )
   END_RUNG
   RUNG wire#w1
      I_Contact( "Unit1.Em2.ControlNodes".cmSuctionPadTopRightVaccum.monitoring.inHomePos )
   END_RUNG wire#w2
   RUNG wire#w1
      I_Contact( "Unit1.Em2.ControlNodes".cmSuctionPadBtmLeftVaccum.monitoring.inHomePos )
   END_RUNG wire#w2
   RUNG wire#w1
      I_Contact( "Unit1.Em2.ControlNodes".cmSuctionPadBtmRightVaccum.monitoring.inHomePos )
   END_RUNG wire#w2
   RUNG wire#w1
      Contact( "Unit1.Em2.ControlNodes".cmSuctionPadTopLeftVaccum.monitoring.inHomePos )
      Contact( "Unit1.Em2.ControlNodes".cmSuctionPadTopRightVaccum.monitoring.inHomePos )
      Contact( "Unit1.Em2.ControlNodes".cmSuctionPadBtmLeftVaccum.monitoring.inHomePos )
      Contact( "Unit1.Em2.ControlNodes".cmSuctionPadBtmRightVaccum.monitoring.inHomePos )
      Coil( "Unit1.Em2.ControlNodes".semiAutoSplice."step".transition1[401] )
   END_RUNG
   RUNG wire#w1
      Contact( "Unit1.Em2.ControlNodes".semiAutoSplice."step".transition1[401] )
      { S7_Templates := "time_type := Time" } #statTonTimer[401].TON(pt := #SeqDelayTime, et =>)
      Move(in := #JOB_4_STEP_02, out1 => "Unit1.Em2.ControlNodes".semiAutoSplice.sequence.status.nextStep)
   END_RUNG
   // the same network as SCL:
   #_w1 := ("Unit1.Em2.ControlNodes".semiAutoSplice.sequence.status.currentStep = #JOB_4_STEP_01) AND "Unit1.Em2.ControlNodes".semiAutoSplice.sequence.status.seqActive;
   "Unit1.Em2.ControlNodes".semiAutoSplice."step".action1[401] := #_w1 AND (NOT "Unit1.Em2.ControlNodes".cmSuctionPadTopLeftVaccum.monitoring.inHomePos OR NOT "Unit1.Em2.ControlNodes".cmSuctionPadTopRightVaccum.monitoring.inHomePos OR NOT "Unit1.Em2.ControlNodes".cmSuctionPadBtmLeftVaccum.monitoring.inHomePos OR NOT "Unit1.Em2.ControlNodes".cmSuctionPadBtmRightVaccum.monitoring.inHomePos);
   "Unit1.Em2.ControlNodes".semiAutoSplice."step".transition1[401] := #_w1 AND "Unit1.Em2.ControlNodes".cmSuctionPadTopLeftVaccum.monitoring.inHomePos AND "Unit1.Em2.ControlNodes".cmSuctionPadTopRightVaccum.monitoring.inHomePos AND "Unit1.Em2.ControlNodes".cmSuctionPadBtmLeftVaccum.monitoring.inHomePos AND "Unit1.Em2.ControlNodes".cmSuctionPadBtmRightVaccum.monitoring.inHomePos;
   #statTonTimer[401].TON(IN := #_w1 AND "Unit1.Em2.ControlNodes".semiAutoSplice."step".transition1[401],
                          PT := #SeqDelayTime);
   IF #statTonTimer[401].Q THEN
       "Unit1.Em2.ControlNodes".semiAutoSplice.sequence.status.nextStep := #JOB_4_STEP_02;
   END_IF;
END_REGION

REGION Network 27: Step[402] :
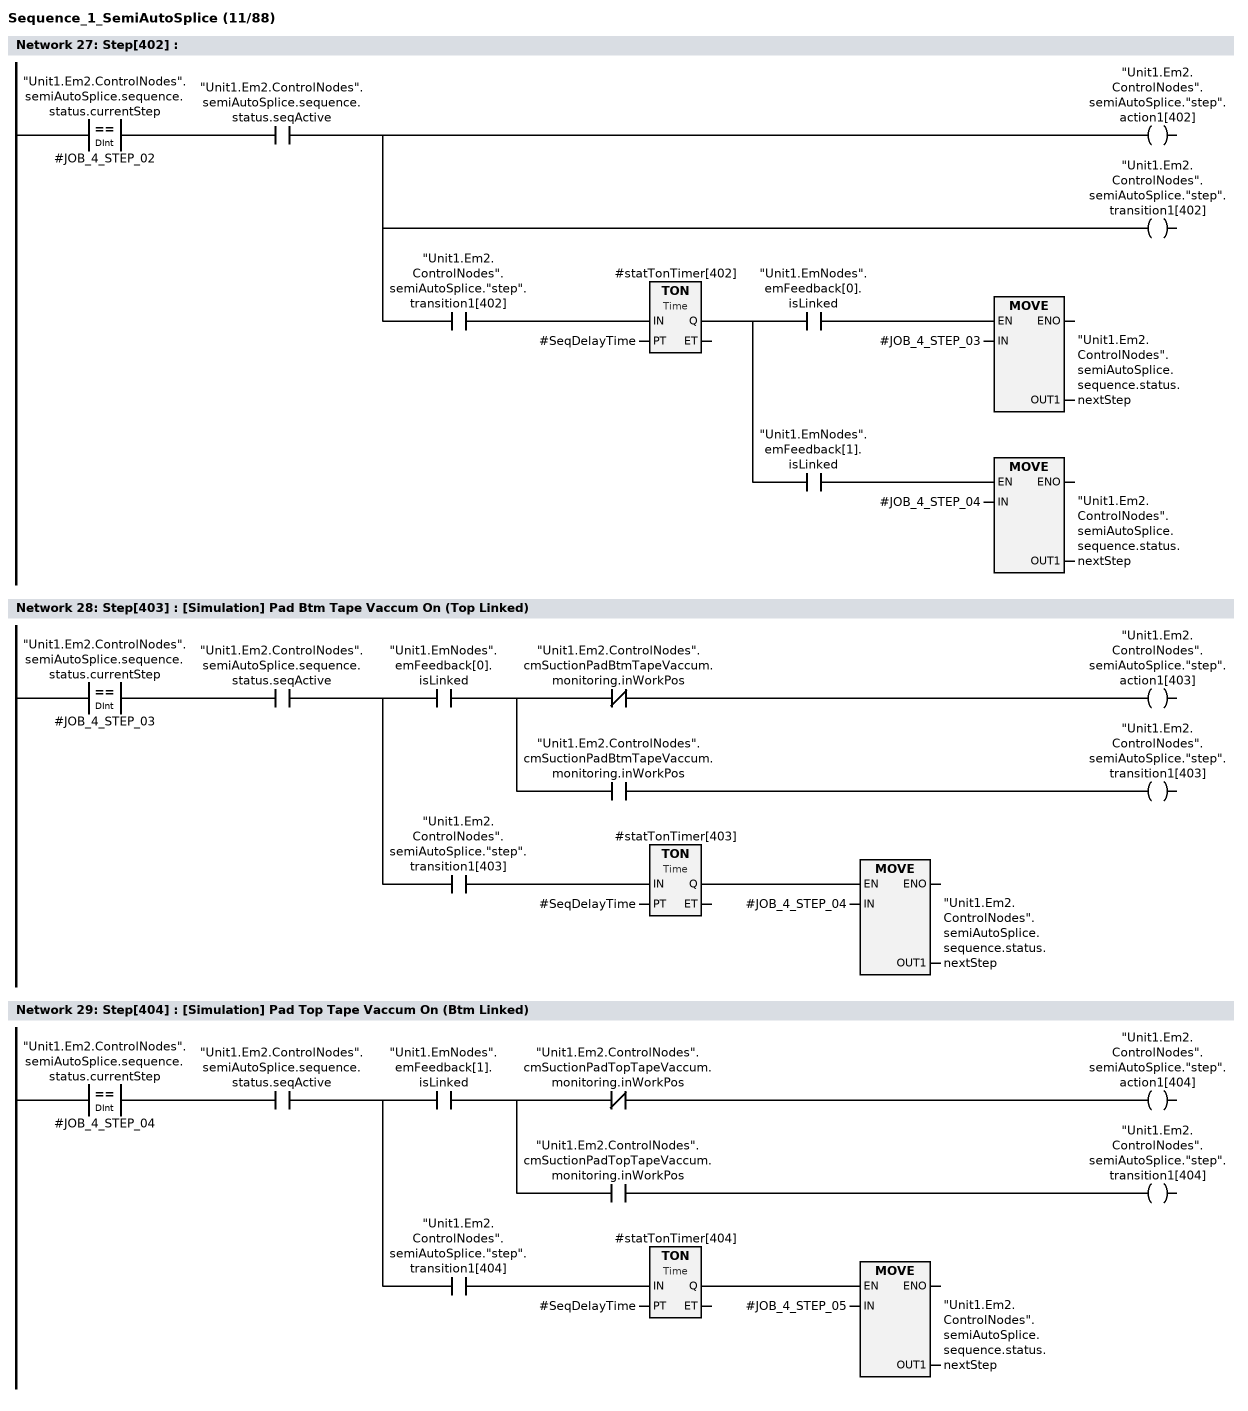
   RUNG wire#powerrail
      { S7_Templates := "SrcType := DInt" } EQ_Contact(in1 := "Unit1.Em2.ControlNodes".semiAutoSplice.sequence.status.currentStep, in2 := #JOB_4_STEP_02)
      Contact( "Unit1.Em2.ControlNodes".semiAutoSplice.sequence.status.seqActive )
      wire#w1
      Coil( "Unit1.Em2.ControlNodes".semiAutoSplice."step".action1[402] )
   END_RUNG
   RUNG wire#w1
      Coil( "Unit1.Em2.ControlNodes".semiAutoSplice."step".transition1[402] )
   END_RUNG
   RUNG wire#w1
      Contact( "Unit1.Em2.ControlNodes".semiAutoSplice."step".transition1[402] )
      { S7_Templates := "time_type := Time" } #statTonTimer[402].TON(pt := #SeqDelayTime, et =>)
      wire#w2
      Contact( "Unit1.EmNodes".emFeedback[0].isLinked )
      Move(in := #JOB_4_STEP_03, out1 => "Unit1.Em2.ControlNodes".semiAutoSplice.sequence.status.nextStep)
   END_RUNG
   RUNG wire#w2
      Contact( "Unit1.EmNodes".emFeedback[1].isLinked )
      Move(in := #JOB_4_STEP_04, out1 => "Unit1.Em2.ControlNodes".semiAutoSplice.sequence.status.nextStep)
   END_RUNG
   // the same network as SCL:
   "Unit1.Em2.ControlNodes".semiAutoSplice."step".action1[402] := ("Unit1.Em2.ControlNodes".semiAutoSplice.sequence.status.currentStep = #JOB_4_STEP_02) AND "Unit1.Em2.ControlNodes".semiAutoSplice.sequence.status.seqActive;
   "Unit1.Em2.ControlNodes".semiAutoSplice."step".transition1[402] := ("Unit1.Em2.ControlNodes".semiAutoSplice.sequence.status.currentStep = #JOB_4_STEP_02) AND "Unit1.Em2.ControlNodes".semiAutoSplice.sequence.status.seqActive;
   #statTonTimer[402].TON(IN := ("Unit1.Em2.ControlNodes".semiAutoSplice.sequence.status.currentStep = #JOB_4_STEP_02) AND "Unit1.Em2.ControlNodes".semiAutoSplice.sequence.status.seqActive AND "Unit1.Em2.ControlNodes".semiAutoSplice."step".transition1[402],
                          PT := #SeqDelayTime);
   IF #statTonTimer[402].Q AND "Unit1.EmNodes".emFeedback[0].isLinked THEN
       "Unit1.Em2.ControlNodes".semiAutoSplice.sequence.status.nextStep := #JOB_4_STEP_03;
   END_IF;
   IF #statTonTimer[402].Q AND "Unit1.EmNodes".emFeedback[1].isLinked THEN
       "Unit1.Em2.ControlNodes".semiAutoSplice.sequence.status.nextStep := #JOB_4_STEP_04;
   END_IF;
END_REGION

REGION Network 28: Step[403] : [Simulation] Pad Btm Tape Vaccum On (Top Linked)
   RUNG wire#powerrail
      { S7_Templates := "SrcType := DInt" } EQ_Contact(in1 := "Unit1.Em2.ControlNodes".semiAutoSplice.sequence.status.currentStep, in2 := #JOB_4_STEP_03)
      Contact( "Unit1.Em2.ControlNodes".semiAutoSplice.sequence.status.seqActive )
      wire#w1
      Contact( "Unit1.EmNodes".emFeedback[0].isLinked )
      wire#w2
      I_Contact( "Unit1.Em2.ControlNodes".cmSuctionPadBtmTapeVaccum.monitoring.inWorkPos )
      Coil( "Unit1.Em2.ControlNodes".semiAutoSplice."step".action1[403] )
   END_RUNG
   RUNG wire#w2
      Contact( "Unit1.Em2.ControlNodes".cmSuctionPadBtmTapeVaccum.monitoring.inWorkPos )
      Coil( "Unit1.Em2.ControlNodes".semiAutoSplice."step".transition1[403] )
   END_RUNG
   RUNG wire#w1
      Contact( "Unit1.Em2.ControlNodes".semiAutoSplice."step".transition1[403] )
      { S7_Templates := "time_type := Time" } #statTonTimer[403].TON(pt := #SeqDelayTime, et =>)
      Move(in := #JOB_4_STEP_04, out1 => "Unit1.Em2.ControlNodes".semiAutoSplice.sequence.status.nextStep)
   END_RUNG
   // the same network as SCL:
   #_w1 := ("Unit1.Em2.ControlNodes".semiAutoSplice.sequence.status.currentStep = #JOB_4_STEP_03) AND "Unit1.Em2.ControlNodes".semiAutoSplice.sequence.status.seqActive;
   #_w2 := #_w1 AND "Unit1.EmNodes".emFeedback[0].isLinked;
   "Unit1.Em2.ControlNodes".semiAutoSplice."step".action1[403] := #_w2 AND NOT "Unit1.Em2.ControlNodes".cmSuctionPadBtmTapeVaccum.monitoring.inWorkPos;
   "Unit1.Em2.ControlNodes".semiAutoSplice."step".transition1[403] := #_w2 AND "Unit1.Em2.ControlNodes".cmSuctionPadBtmTapeVaccum.monitoring.inWorkPos;
   #statTonTimer[403].TON(IN := #_w1 AND "Unit1.Em2.ControlNodes".semiAutoSplice."step".transition1[403],
                          PT := #SeqDelayTime);
   IF #statTonTimer[403].Q THEN
       "Unit1.Em2.ControlNodes".semiAutoSplice.sequence.status.nextStep := #JOB_4_STEP_04;
   END_IF;
END_REGION

REGION Network 29: Step[404] : [Simulation] Pad Top Tape Vaccum On (Btm Linked)
   RUNG wire#powerrail
      { S7_Templates := "SrcType := DInt" } EQ_Contact(in1 := "Unit1.Em2.ControlNodes".semiAutoSplice.sequence.status.currentStep, in2 := #JOB_4_STEP_04)
      Contact( "Unit1.Em2.ControlNodes".semiAutoSplice.sequence.status.seqActive )
      wire#w1
      Contact( "Unit1.EmNodes".emFeedback[1].isLinked )
      wire#w2
      I_Contact( "Unit1.Em2.ControlNodes".cmSuctionPadTopTapeVaccum.monitoring.inWorkPos )
      Coil( "Unit1.Em2.ControlNodes".semiAutoSplice."step".action1[404] )
   END_RUNG
   RUNG wire#w2
      Contact( "Unit1.Em2.ControlNodes".cmSuctionPadTopTapeVaccum.monitoring.inWorkPos )
      Coil( "Unit1.Em2.ControlNodes".semiAutoSplice."step".transition1[404] )
   END_RUNG
   RUNG wire#w1
      Contact( "Unit1.Em2.ControlNodes".semiAutoSplice."step".transition1[404] )
      { S7_Templates := "time_type := Time" } #statTonTimer[404].TON(pt := #SeqDelayTime, et =>)
      Move(in := #JOB_4_STEP_05, out1 => "Unit1.Em2.ControlNodes".semiAutoSplice.sequence.status.nextStep)
   END_RUNG
   // the same network as SCL:
   #_w1 := ("Unit1.Em2.ControlNodes".semiAutoSplice.sequence.status.currentStep = #JOB_4_STEP_04) AND "Unit1.Em2.ControlNodes".semiAutoSplice.sequence.status.seqActive;
   #_w2 := #_w1 AND "Unit1.EmNodes".emFeedback[1].isLinked;
   "Unit1.Em2.ControlNodes".semiAutoSplice."step".action1[404] := #_w2 AND NOT "Unit1.Em2.ControlNodes".cmSuctionPadTopTapeVaccum.monitoring.inWorkPos;
   "Unit1.Em2.ControlNodes".semiAutoSplice."step".transition1[404] := #_w2 AND "Unit1.Em2.ControlNodes".cmSuctionPadTopTapeVaccum.monitoring.inWorkPos;
   #statTonTimer[404].TON(IN := #_w1 AND "Unit1.Em2.ControlNodes".semiAutoSplice."step".transition1[404],
                          PT := #SeqDelayTime);
   IF #statTonTimer[404].Q THEN
       "Unit1.Em2.ControlNodes".semiAutoSplice.sequence.status.nextStep := #JOB_4_STEP_05;
   END_IF;
END_REGION

REGION Network 30: Step[405] : cutter home (Down)
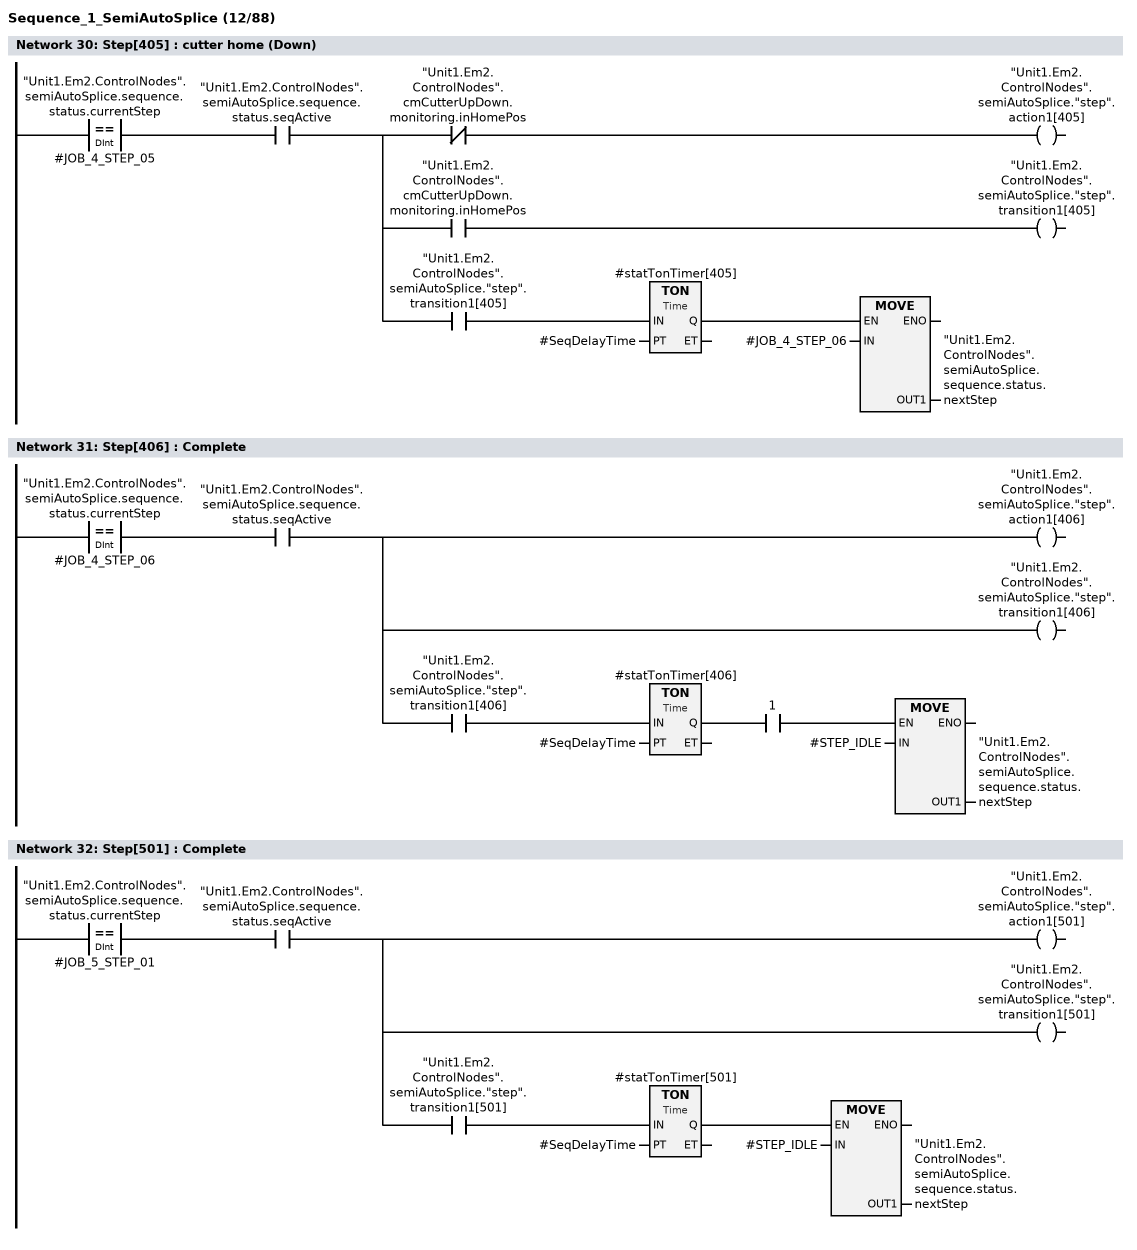
   RUNG wire#powerrail
      { S7_Templates := "SrcType := DInt" } EQ_Contact(in1 := "Unit1.Em2.ControlNodes".semiAutoSplice.sequence.status.currentStep, in2 := #JOB_4_STEP_05)
      Contact( "Unit1.Em2.ControlNodes".semiAutoSplice.sequence.status.seqActive )
      wire#w1
      I_Contact( "Unit1.Em2.ControlNodes".cmCutterUpDown.monitoring.inHomePos )
      Coil( "Unit1.Em2.ControlNodes".semiAutoSplice."step".action1[405] )
   END_RUNG
   RUNG wire#w1
      Contact( "Unit1.Em2.ControlNodes".cmCutterUpDown.monitoring.inHomePos )
      Coil( "Unit1.Em2.ControlNodes".semiAutoSplice."step".transition1[405] )
   END_RUNG
   RUNG wire#w1
      Contact( "Unit1.Em2.ControlNodes".semiAutoSplice."step".transition1[405] )
      { S7_Templates := "time_type := Time" } #statTonTimer[405].TON(pt := #SeqDelayTime, et =>)
      Move(in := #JOB_4_STEP_06, out1 => "Unit1.Em2.ControlNodes".semiAutoSplice.sequence.status.nextStep)
   END_RUNG
   // the same network as SCL:
   #_w1 := ("Unit1.Em2.ControlNodes".semiAutoSplice.sequence.status.currentStep = #JOB_4_STEP_05) AND "Unit1.Em2.ControlNodes".semiAutoSplice.sequence.status.seqActive;
   "Unit1.Em2.ControlNodes".semiAutoSplice."step".action1[405] := #_w1 AND NOT "Unit1.Em2.ControlNodes".cmCutterUpDown.monitoring.inHomePos;
   "Unit1.Em2.ControlNodes".semiAutoSplice."step".transition1[405] := #_w1 AND "Unit1.Em2.ControlNodes".cmCutterUpDown.monitoring.inHomePos;
   #statTonTimer[405].TON(IN := #_w1 AND "Unit1.Em2.ControlNodes".semiAutoSplice."step".transition1[405],
                          PT := #SeqDelayTime);
   IF #statTonTimer[405].Q THEN
       "Unit1.Em2.ControlNodes".semiAutoSplice.sequence.status.nextStep := #JOB_4_STEP_06;
   END_IF;
END_REGION

REGION Network 31: Step[406] : Complete
   RUNG wire#powerrail
      { S7_Templates := "SrcType := DInt" } EQ_Contact(in1 := "Unit1.Em2.ControlNodes".semiAutoSplice.sequence.status.currentStep, in2 := #JOB_4_STEP_06)
      Contact( "Unit1.Em2.ControlNodes".semiAutoSplice.sequence.status.seqActive )
      wire#w1
      Coil( "Unit1.Em2.ControlNodes".semiAutoSplice."step".action1[406] )
   END_RUNG
   RUNG wire#w1
      Coil( "Unit1.Em2.ControlNodes".semiAutoSplice."step".transition1[406] )
   END_RUNG
   RUNG wire#w1
      Contact( "Unit1.Em2.ControlNodes".semiAutoSplice."step".transition1[406] )
      { S7_Templates := "time_type := Time" } #statTonTimer[406].TON(pt := #SeqDelayTime, et =>)
      Contact( 1 )
      Move(in := #STEP_IDLE, out1 => "Unit1.Em2.ControlNodes".semiAutoSplice.sequence.status.nextStep)
   END_RUNG
   // the same network as SCL:
   "Unit1.Em2.ControlNodes".semiAutoSplice."step".action1[406] := ("Unit1.Em2.ControlNodes".semiAutoSplice.sequence.status.currentStep = #JOB_4_STEP_06) AND "Unit1.Em2.ControlNodes".semiAutoSplice.sequence.status.seqActive;
   "Unit1.Em2.ControlNodes".semiAutoSplice."step".transition1[406] := ("Unit1.Em2.ControlNodes".semiAutoSplice.sequence.status.currentStep = #JOB_4_STEP_06) AND "Unit1.Em2.ControlNodes".semiAutoSplice.sequence.status.seqActive;
   #statTonTimer[406].TON(IN := ("Unit1.Em2.ControlNodes".semiAutoSplice.sequence.status.currentStep = #JOB_4_STEP_06) AND "Unit1.Em2.ControlNodes".semiAutoSplice.sequence.status.seqActive AND "Unit1.Em2.ControlNodes".semiAutoSplice."step".transition1[406],
                          PT := #SeqDelayTime);
   IF #statTonTimer[406].Q AND 1 THEN
       "Unit1.Em2.ControlNodes".semiAutoSplice.sequence.status.nextStep := #STEP_IDLE;
   END_IF;
END_REGION

REGION Network 32: Step[501] : Complete
   RUNG wire#powerrail
      { S7_Templates := "SrcType := DInt" } EQ_Contact(in1 := "Unit1.Em2.ControlNodes".semiAutoSplice.sequence.status.currentStep, in2 := #JOB_5_STEP_01)
      Contact( "Unit1.Em2.ControlNodes".semiAutoSplice.sequence.status.seqActive )
      wire#w1
      Coil( "Unit1.Em2.ControlNodes".semiAutoSplice."step".action1[501] )
   END_RUNG
   RUNG wire#w1
      Coil( "Unit1.Em2.ControlNodes".semiAutoSplice."step".transition1[501] )
   END_RUNG
   RUNG wire#w1
      Contact( "Unit1.Em2.ControlNodes".semiAutoSplice."step".transition1[501] )
      { S7_Templates := "time_type := Time" } #statTonTimer[501].TON(pt := #SeqDelayTime, et =>)
      Move(in := #STEP_IDLE, out1 => "Unit1.Em2.ControlNodes".semiAutoSplice.sequence.status.nextStep)
   END_RUNG
   // the same network as SCL:
   "Unit1.Em2.ControlNodes".semiAutoSplice."step".action1[501] := ("Unit1.Em2.ControlNodes".semiAutoSplice.sequence.status.currentStep = #JOB_5_STEP_01) AND "Unit1.Em2.ControlNodes".semiAutoSplice.sequence.status.seqActive;
   "Unit1.Em2.ControlNodes".semiAutoSplice."step".transition1[501] := ("Unit1.Em2.ControlNodes".semiAutoSplice.sequence.status.currentStep = #JOB_5_STEP_01) AND "Unit1.Em2.ControlNodes".semiAutoSplice.sequence.status.seqActive;
   #statTonTimer[501].TON(IN := ("Unit1.Em2.ControlNodes".semiAutoSplice.sequence.status.currentStep = #JOB_5_STEP_01) AND "Unit1.Em2.ControlNodes".semiAutoSplice.sequence.status.seqActive AND "Unit1.Em2.ControlNodes".semiAutoSplice."step".transition1[501],
                          PT := #SeqDelayTime);
   IF #statTonTimer[501].Q THEN
       "Unit1.Em2.ControlNodes".semiAutoSplice.sequence.status.nextStep := #STEP_IDLE;
   END_IF;
END_REGION

REGION Network 33: Step[601] : diameter check & Link/Unlink & Pad Top/Btm Work (Up)
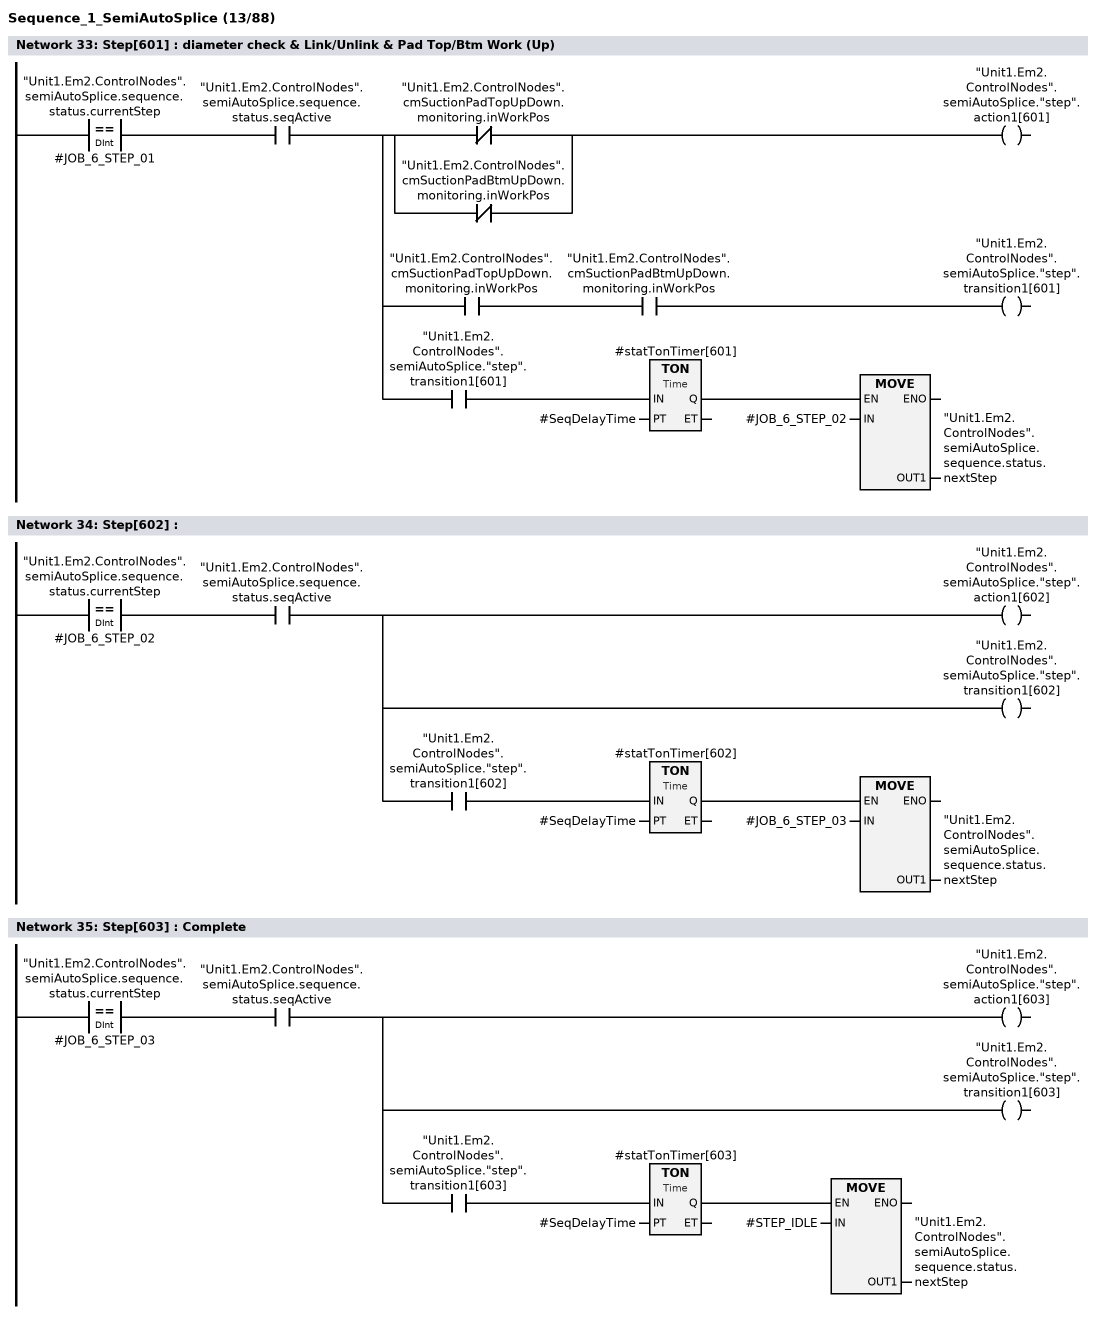
   RUNG wire#powerrail
      { S7_Templates := "SrcType := DInt" } EQ_Contact(in1 := "Unit1.Em2.ControlNodes".semiAutoSplice.sequence.status.currentStep, in2 := #JOB_6_STEP_01)
      Contact( "Unit1.Em2.ControlNodes".semiAutoSplice.sequence.status.seqActive )
      wire#w1
      I_Contact( "Unit1.Em2.ControlNodes".cmSuctionPadTopUpDown.monitoring.inWorkPos )
      wire#w2
      Coil( "Unit1.Em2.ControlNodes".semiAutoSplice."step".action1[601] )
   END_RUNG
   RUNG wire#w1
      I_Contact( "Unit1.Em2.ControlNodes".cmSuctionPadBtmUpDown.monitoring.inWorkPos )
   END_RUNG wire#w2
   RUNG wire#w1
      Contact( "Unit1.Em2.ControlNodes".cmSuctionPadTopUpDown.monitoring.inWorkPos )
      Contact( "Unit1.Em2.ControlNodes".cmSuctionPadBtmUpDown.monitoring.inWorkPos )
      Coil( "Unit1.Em2.ControlNodes".semiAutoSplice."step".transition1[601] )
   END_RUNG
   RUNG wire#w1
      Contact( "Unit1.Em2.ControlNodes".semiAutoSplice."step".transition1[601] )
      { S7_Templates := "time_type := Time" } #statTonTimer[601].TON(pt := #SeqDelayTime, et =>)
      Move(in := #JOB_6_STEP_02, out1 => "Unit1.Em2.ControlNodes".semiAutoSplice.sequence.status.nextStep)
   END_RUNG
   // the same network as SCL:
   #_w1 := ("Unit1.Em2.ControlNodes".semiAutoSplice.sequence.status.currentStep = #JOB_6_STEP_01) AND "Unit1.Em2.ControlNodes".semiAutoSplice.sequence.status.seqActive;
   "Unit1.Em2.ControlNodes".semiAutoSplice."step".action1[601] := #_w1 AND (NOT "Unit1.Em2.ControlNodes".cmSuctionPadTopUpDown.monitoring.inWorkPos OR NOT "Unit1.Em2.ControlNodes".cmSuctionPadBtmUpDown.monitoring.inWorkPos);
   "Unit1.Em2.ControlNodes".semiAutoSplice."step".transition1[601] := #_w1 AND "Unit1.Em2.ControlNodes".cmSuctionPadTopUpDown.monitoring.inWorkPos AND "Unit1.Em2.ControlNodes".cmSuctionPadBtmUpDown.monitoring.inWorkPos;
   #statTonTimer[601].TON(IN := #_w1 AND "Unit1.Em2.ControlNodes".semiAutoSplice."step".transition1[601],
                          PT := #SeqDelayTime);
   IF #statTonTimer[601].Q THEN
       "Unit1.Em2.ControlNodes".semiAutoSplice.sequence.status.nextStep := #JOB_6_STEP_02;
   END_IF;
END_REGION

REGION Network 34: Step[602] :
   RUNG wire#powerrail
      { S7_Templates := "SrcType := DInt" } EQ_Contact(in1 := "Unit1.Em2.ControlNodes".semiAutoSplice.sequence.status.currentStep, in2 := #JOB_6_STEP_02)
      Contact( "Unit1.Em2.ControlNodes".semiAutoSplice.sequence.status.seqActive )
      wire#w1
      Coil( "Unit1.Em2.ControlNodes".semiAutoSplice."step".action1[602] )
   END_RUNG
   RUNG wire#w1
      Coil( "Unit1.Em2.ControlNodes".semiAutoSplice."step".transition1[602] )
   END_RUNG
   RUNG wire#w1
      Contact( "Unit1.Em2.ControlNodes".semiAutoSplice."step".transition1[602] )
      { S7_Templates := "time_type := Time" } #statTonTimer[602].TON(pt := #SeqDelayTime, et =>)
      Move(in := #JOB_6_STEP_03, out1 => "Unit1.Em2.ControlNodes".semiAutoSplice.sequence.status.nextStep)
   END_RUNG
   // the same network as SCL:
   "Unit1.Em2.ControlNodes".semiAutoSplice."step".action1[602] := ("Unit1.Em2.ControlNodes".semiAutoSplice.sequence.status.currentStep = #JOB_6_STEP_02) AND "Unit1.Em2.ControlNodes".semiAutoSplice.sequence.status.seqActive;
   "Unit1.Em2.ControlNodes".semiAutoSplice."step".transition1[602] := ("Unit1.Em2.ControlNodes".semiAutoSplice.sequence.status.currentStep = #JOB_6_STEP_02) AND "Unit1.Em2.ControlNodes".semiAutoSplice.sequence.status.seqActive;
   #statTonTimer[602].TON(IN := ("Unit1.Em2.ControlNodes".semiAutoSplice.sequence.status.currentStep = #JOB_6_STEP_02) AND "Unit1.Em2.ControlNodes".semiAutoSplice.sequence.status.seqActive AND "Unit1.Em2.ControlNodes".semiAutoSplice."step".transition1[602],
                          PT := #SeqDelayTime);
   IF #statTonTimer[602].Q THEN
       "Unit1.Em2.ControlNodes".semiAutoSplice.sequence.status.nextStep := #JOB_6_STEP_03;
   END_IF;
END_REGION

REGION Network 35: Step[603] : Complete
   RUNG wire#powerrail
      { S7_Templates := "SrcType := DInt" } EQ_Contact(in1 := "Unit1.Em2.ControlNodes".semiAutoSplice.sequence.status.currentStep, in2 := #JOB_6_STEP_03)
      Contact( "Unit1.Em2.ControlNodes".semiAutoSplice.sequence.status.seqActive )
      wire#w1
      Coil( "Unit1.Em2.ControlNodes".semiAutoSplice."step".action1[603] )
   END_RUNG
   RUNG wire#w1
      Coil( "Unit1.Em2.ControlNodes".semiAutoSplice."step".transition1[603] )
   END_RUNG
   RUNG wire#w1
      Contact( "Unit1.Em2.ControlNodes".semiAutoSplice."step".transition1[603] )
      { S7_Templates := "time_type := Time" } #statTonTimer[603].TON(pt := #SeqDelayTime, et =>)
      Move(in := #STEP_IDLE, out1 => "Unit1.Em2.ControlNodes".semiAutoSplice.sequence.status.nextStep)
   END_RUNG
   // the same network as SCL:
   "Unit1.Em2.ControlNodes".semiAutoSplice."step".action1[603] := ("Unit1.Em2.ControlNodes".semiAutoSplice.sequence.status.currentStep = #JOB_6_STEP_03) AND "Unit1.Em2.ControlNodes".semiAutoSplice.sequence.status.seqActive;
   "Unit1.Em2.ControlNodes".semiAutoSplice."step".transition1[603] := ("Unit1.Em2.ControlNodes".semiAutoSplice.sequence.status.currentStep = #JOB_6_STEP_03) AND "Unit1.Em2.ControlNodes".semiAutoSplice.sequence.status.seqActive;
   #statTonTimer[603].TON(IN := ("Unit1.Em2.ControlNodes".semiAutoSplice.sequence.status.currentStep = #JOB_6_STEP_03) AND "Unit1.Em2.ControlNodes".semiAutoSplice.sequence.status.seqActive AND "Unit1.Em2.ControlNodes".semiAutoSplice."step".transition1[603],
                          PT := #SeqDelayTime);
   IF #statTonTimer[603].Q THEN
       "Unit1.Em2.ControlNodes".semiAutoSplice.sequence.status.nextStep := #STEP_IDLE;
   END_IF;
END_REGION

REGION Network 36: Step[701] : Pad Top/Btm Left/Right Vacc On
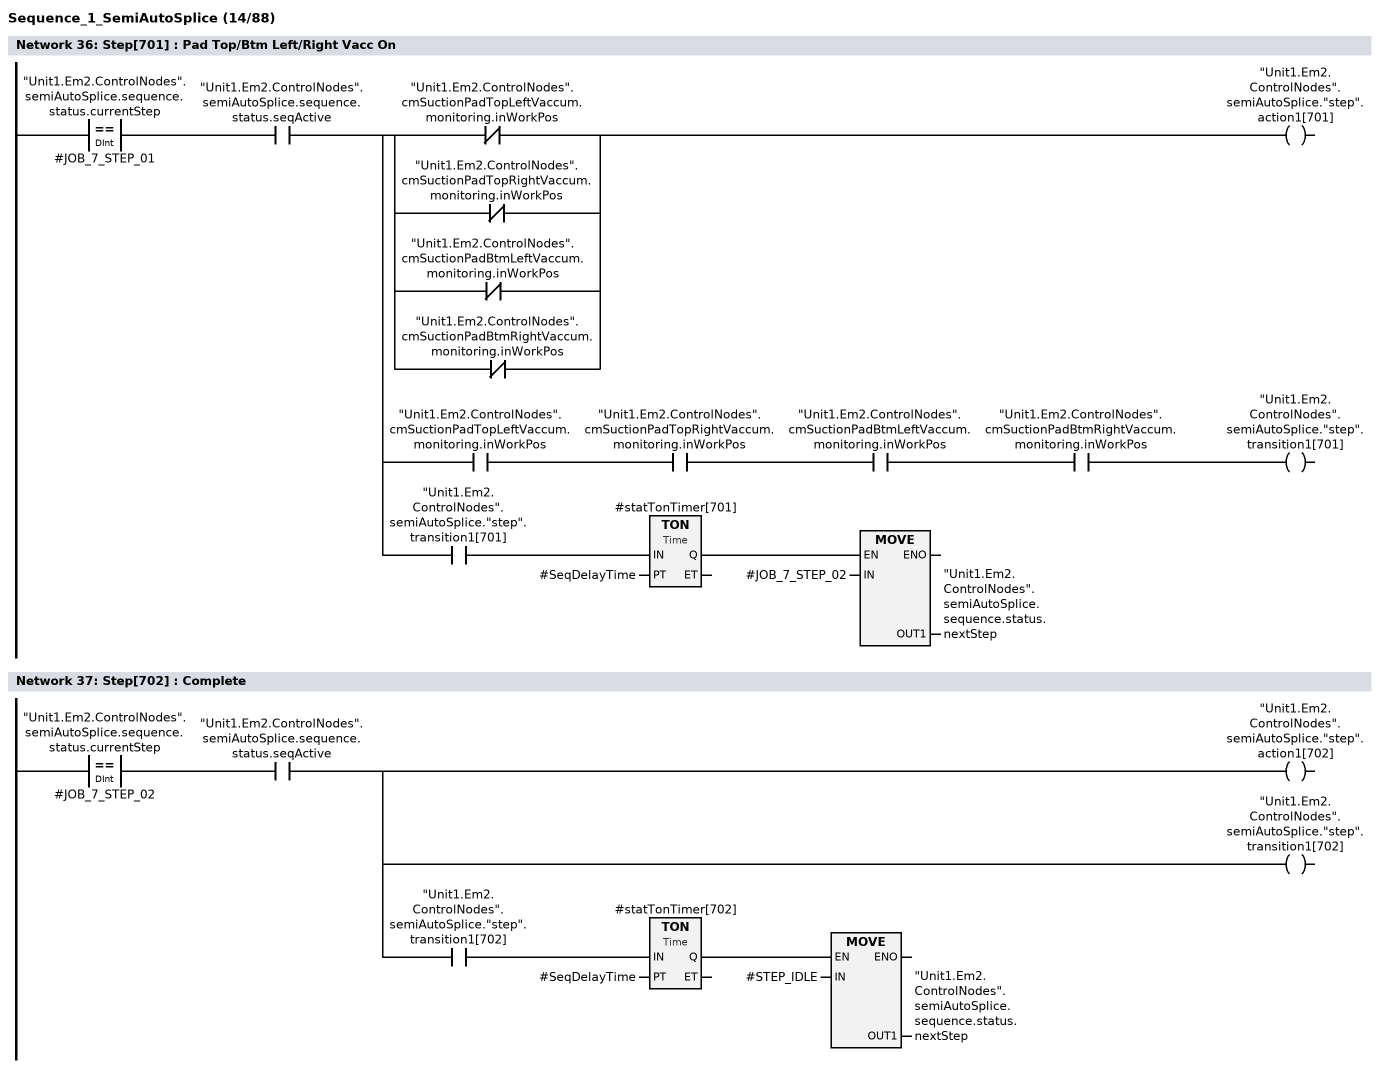
   RUNG wire#powerrail
      { S7_Templates := "SrcType := DInt" } EQ_Contact(in1 := "Unit1.Em2.ControlNodes".semiAutoSplice.sequence.status.currentStep, in2 := #JOB_7_STEP_01)
      Contact( "Unit1.Em2.ControlNodes".semiAutoSplice.sequence.status.seqActive )
      wire#w1
      I_Contact( "Unit1.Em2.ControlNodes".cmSuctionPadTopLeftVaccum.monitoring.inWorkPos )
      wire#w2
      Coil( "Unit1.Em2.ControlNodes".semiAutoSplice."step".action1[701] )
   END_RUNG
   RUNG wire#w1
      I_Contact( "Unit1.Em2.ControlNodes".cmSuctionPadTopRightVaccum.monitoring.inWorkPos )
   END_RUNG wire#w2
   RUNG wire#w1
      I_Contact( "Unit1.Em2.ControlNodes".cmSuctionPadBtmLeftVaccum.monitoring.inWorkPos )
   END_RUNG wire#w2
   RUNG wire#w1
      I_Contact( "Unit1.Em2.ControlNodes".cmSuctionPadBtmRightVaccum.monitoring.inWorkPos )
   END_RUNG wire#w2
   RUNG wire#w1
      Contact( "Unit1.Em2.ControlNodes".cmSuctionPadTopLeftVaccum.monitoring.inWorkPos )
      Contact( "Unit1.Em2.ControlNodes".cmSuctionPadTopRightVaccum.monitoring.inWorkPos )
      Contact( "Unit1.Em2.ControlNodes".cmSuctionPadBtmLeftVaccum.monitoring.inWorkPos )
      Contact( "Unit1.Em2.ControlNodes".cmSuctionPadBtmRightVaccum.monitoring.inWorkPos )
      Coil( "Unit1.Em2.ControlNodes".semiAutoSplice."step".transition1[701] )
   END_RUNG
   RUNG wire#w1
      Contact( "Unit1.Em2.ControlNodes".semiAutoSplice."step".transition1[701] )
      { S7_Templates := "time_type := Time" } #statTonTimer[701].TON(pt := #SeqDelayTime, et =>)
      Move(in := #JOB_7_STEP_02, out1 => "Unit1.Em2.ControlNodes".semiAutoSplice.sequence.status.nextStep)
   END_RUNG
   // the same network as SCL:
   #_w1 := ("Unit1.Em2.ControlNodes".semiAutoSplice.sequence.status.currentStep = #JOB_7_STEP_01) AND "Unit1.Em2.ControlNodes".semiAutoSplice.sequence.status.seqActive;
   "Unit1.Em2.ControlNodes".semiAutoSplice."step".action1[701] := #_w1 AND (NOT "Unit1.Em2.ControlNodes".cmSuctionPadTopLeftVaccum.monitoring.inWorkPos OR NOT "Unit1.Em2.ControlNodes".cmSuctionPadTopRightVaccum.monitoring.inWorkPos OR NOT "Unit1.Em2.ControlNodes".cmSuctionPadBtmLeftVaccum.monitoring.inWorkPos OR NOT "Unit1.Em2.ControlNodes".cmSuctionPadBtmRightVaccum.monitoring.inWorkPos);
   "Unit1.Em2.ControlNodes".semiAutoSplice."step".transition1[701] := #_w1 AND "Unit1.Em2.ControlNodes".cmSuctionPadTopLeftVaccum.monitoring.inWorkPos AND "Unit1.Em2.ControlNodes".cmSuctionPadTopRightVaccum.monitoring.inWorkPos AND "Unit1.Em2.ControlNodes".cmSuctionPadBtmLeftVaccum.monitoring.inWorkPos AND "Unit1.Em2.ControlNodes".cmSuctionPadBtmRightVaccum.monitoring.inWorkPos;
   #statTonTimer[701].TON(IN := #_w1 AND "Unit1.Em2.ControlNodes".semiAutoSplice."step".transition1[701],
                          PT := #SeqDelayTime);
   IF #statTonTimer[701].Q THEN
       "Unit1.Em2.ControlNodes".semiAutoSplice.sequence.status.nextStep := #JOB_7_STEP_02;
   END_IF;
END_REGION

REGION Network 37: Step[702] : Complete
   RUNG wire#powerrail
      { S7_Templates := "SrcType := DInt" } EQ_Contact(in1 := "Unit1.Em2.ControlNodes".semiAutoSplice.sequence.status.currentStep, in2 := #JOB_7_STEP_02)
      Contact( "Unit1.Em2.ControlNodes".semiAutoSplice.sequence.status.seqActive )
      wire#w1
      Coil( "Unit1.Em2.ControlNodes".semiAutoSplice."step".action1[702] )
   END_RUNG
   RUNG wire#w1
      Coil( "Unit1.Em2.ControlNodes".semiAutoSplice."step".transition1[702] )
   END_RUNG
   RUNG wire#w1
      Contact( "Unit1.Em2.ControlNodes".semiAutoSplice."step".transition1[702] )
      { S7_Templates := "time_type := Time" } #statTonTimer[702].TON(pt := #SeqDelayTime, et =>)
      Move(in := #STEP_IDLE, out1 => "Unit1.Em2.ControlNodes".semiAutoSplice.sequence.status.nextStep)
   END_RUNG
   // the same network as SCL:
   "Unit1.Em2.ControlNodes".semiAutoSplice."step".action1[702] := ("Unit1.Em2.ControlNodes".semiAutoSplice.sequence.status.currentStep = #JOB_7_STEP_02) AND "Unit1.Em2.ControlNodes".semiAutoSplice.sequence.status.seqActive;
   "Unit1.Em2.ControlNodes".semiAutoSplice."step".transition1[702] := ("Unit1.Em2.ControlNodes".semiAutoSplice.sequence.status.currentStep = #JOB_7_STEP_02) AND "Unit1.Em2.ControlNodes".semiAutoSplice.sequence.status.seqActive;
   #statTonTimer[702].TON(IN := ("Unit1.Em2.ControlNodes".semiAutoSplice.sequence.status.currentStep = #JOB_7_STEP_02) AND "Unit1.Em2.ControlNodes".semiAutoSplice.sequence.status.seqActive AND "Unit1.Em2.ControlNodes".semiAutoSplice."step".transition1[702],
                          PT := #SeqDelayTime);
   IF #statTonTimer[702].Q THEN
       "Unit1.Em2.ControlNodes".semiAutoSplice.sequence.status.nextStep := #STEP_IDLE;
   END_IF;
END_REGION

REGION Network 38: Step[801] : Pad Work & Vacc work, cutter work (Up)
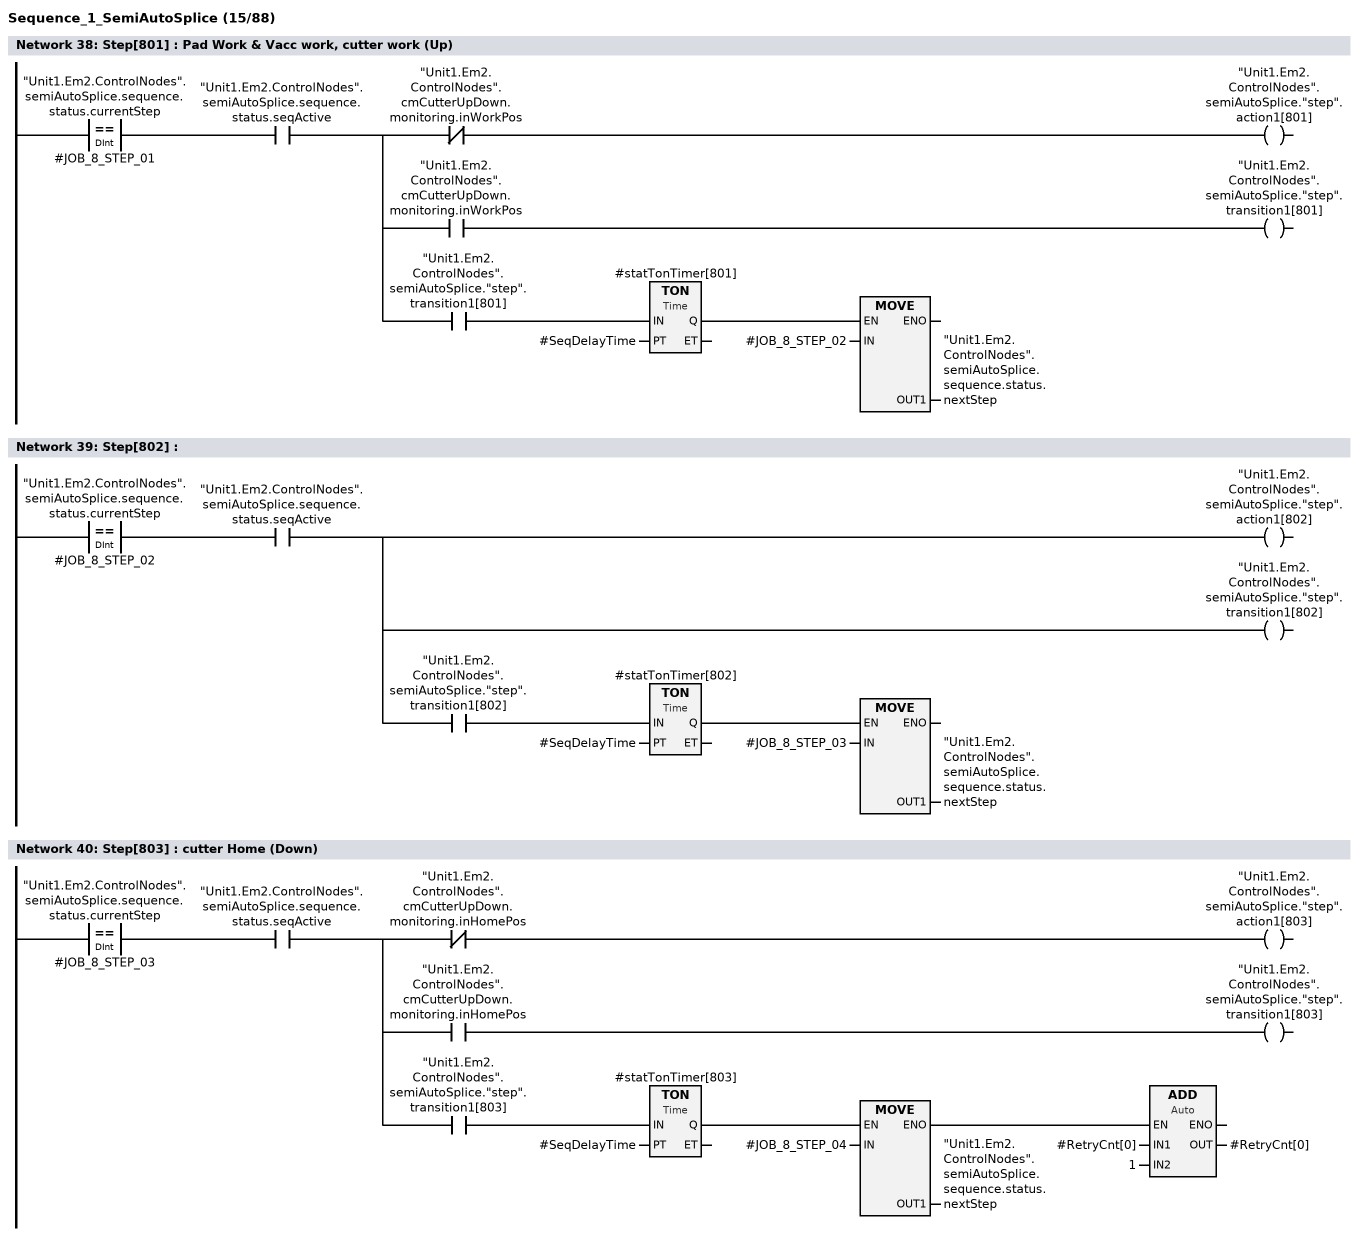
   RUNG wire#powerrail
      { S7_Templates := "SrcType := DInt" } EQ_Contact(in1 := "Unit1.Em2.ControlNodes".semiAutoSplice.sequence.status.currentStep, in2 := #JOB_8_STEP_01)
      Contact( "Unit1.Em2.ControlNodes".semiAutoSplice.sequence.status.seqActive )
      wire#w1
      I_Contact( "Unit1.Em2.ControlNodes".cmCutterUpDown.monitoring.inWorkPos )
      Coil( "Unit1.Em2.ControlNodes".semiAutoSplice."step".action1[801] )
   END_RUNG
   RUNG wire#w1
      Contact( "Unit1.Em2.ControlNodes".cmCutterUpDown.monitoring.inWorkPos )
      Coil( "Unit1.Em2.ControlNodes".semiAutoSplice."step".transition1[801] )
   END_RUNG
   RUNG wire#w1
      Contact( "Unit1.Em2.ControlNodes".semiAutoSplice."step".transition1[801] )
      { S7_Templates := "time_type := Time" } #statTonTimer[801].TON(pt := #SeqDelayTime, et =>)
      Move(in := #JOB_8_STEP_02, out1 => "Unit1.Em2.ControlNodes".semiAutoSplice.sequence.status.nextStep)
   END_RUNG
   // the same network as SCL:
   #_w1 := ("Unit1.Em2.ControlNodes".semiAutoSplice.sequence.status.currentStep = #JOB_8_STEP_01) AND "Unit1.Em2.ControlNodes".semiAutoSplice.sequence.status.seqActive;
   "Unit1.Em2.ControlNodes".semiAutoSplice."step".action1[801] := #_w1 AND NOT "Unit1.Em2.ControlNodes".cmCutterUpDown.monitoring.inWorkPos;
   "Unit1.Em2.ControlNodes".semiAutoSplice."step".transition1[801] := #_w1 AND "Unit1.Em2.ControlNodes".cmCutterUpDown.monitoring.inWorkPos;
   #statTonTimer[801].TON(IN := #_w1 AND "Unit1.Em2.ControlNodes".semiAutoSplice."step".transition1[801],
                          PT := #SeqDelayTime);
   IF #statTonTimer[801].Q THEN
       "Unit1.Em2.ControlNodes".semiAutoSplice.sequence.status.nextStep := #JOB_8_STEP_02;
   END_IF;
END_REGION

